C09120=1115.319,207.001,-67.010,-178.939,9.439,149.564
C09121=1115.314,207.249,-67.035,-178.936,9.442,149.564
C09122=1115.310,207.498,-67.061,-178.933,9.445,149.564
C09123=1115.306,207.747,-67.087,-178.930,9.447,149.564
C09124=1115.301,207.995,-67.112,-178.927,9.450,149.564
C09125=1115.297,208.244,-67.138,-178.925,9.453,149.564
C09126=1115.292,208.493,-67.164,-178.922,9.456,149.564
C09127=1115.288,208.741,-67.190,-178.919,9.459,149.564
C09128=1115.283,208.990,-67.215,-178.916,9.462,149.564
C09129=1115.279,209.238,-67.241,-178.914,9.465,149.564
C09130=1115.275,209.487,-67.266,-178.911,9.468,149.564
C09131=1115.271,209.736,-67.292,-178.908,9.470,149.564
C09132=1115.266,209.984,-67.318,-178.906,9.474,149.564
C09133=1115.262,210.233,-67.343,-178.903,9.476,149.564
C09134=1115.257,210.482,-67.370,-178.900,9.479,149.564
C09135=1115.252,210.731,-67.395,-178.897,9.482,149.563
C09136=1115.248,210.979,-67.421,-178.895,9.485,149.564
C09137=1115.244,211.227,-67.447,-178.892,9.488,149.564
C09138=1115.239,211.476,-67.473,-178.889,9.491,149.563
C09139=1115.235,211.725,-67.499,-178.887,9.494,149.564
C09140=1115.231,211.938,-67.521,-178.884,9.497,149.564
C09141=1115.227,212.151,-67.543,-178.882,9.499,149.563
C09142=1115.224,212.365,-67.565,-178.879,9.502,149.563
C09143=1115.220,212.579,-67.588,-178.877,9.505,149.564
C09144=1115.216,212.791,-67.609,-178.875,9.508,149.564
C09145=1115.212,213.005,-67.632,-178.873,9.510,149.564
C09146=1115.208,213.218,-67.654,-178.870,9.513,149.564
C09147=1115.204,213.432,-67.677,-178.869,9.516,149.564
C09148=1115.199,213.680,-67.703,-178.866,9.519,149.564
C09149=1115.196,213.928,-67.729,-178.864,9.521,149.564
C09150=1115.191,214.177,-67.755,-178.862,9.524,149.564
C09151=1115.187,214.426,-67.781,-178.860,9.527,149.564
C09152=1115.182,214.675,-67.807,-178.858,9.530,149.564
C09153=1115.178,214.923,-67.833,-178.856,9.532,149.564
C09154=1115.174,215.172,-67.859,-178.854,9.536,149.565
C09155=1115.168,215.420,-67.885,-178.851,9.539,149.565
C09156=1115.165,215.668,-67.912,-178.849,9.541,149.565
C09157=1115.160,215.917,-67.937,-178.847,9.544,149.565
C09158=1115.156,216.166,-67.963,-178.845,9.548,149.565
C09159=1115.151,216.415,-67.990,-178.843,9.550,149.565
C09160=1115.147,216.663,-68.016,-178.840,9.553,149.565
C09161=1115.143,216.912,-68.042,-178.838,9.556,149.565
C09162=1115.138,217.161,-68.069,-178.836,9.559,149.565
C09163=1115.134,217.409,-68.094,-178.834,9.562,149.565
C09164=1115.130,217.657,-68.121,-178.831,9.565,149.566
C09165=1115.125,217.906,-68.147,-178.829,9.568,149.566
C09166=1115.121,218.154,-68.173,-178.827,9.571,149.566
C09167=1115.116,218.403,-68.199,-178.825,9.574,149.566
C09168=1115.112,218.652,-68.226,-178.822,9.577,149.566
C09169=1115.108,218.900,-68.252,-178.819,9.580,149.566
C09170=1115.103,219.149,-68.279,-178.817,9.584,149.566
C09171=1115.099,219.398,-68.305,-178.815,9.587,149.566
C09172=1115.095,219.646,-68.331,-178.813,9.589,149.566
C09173=1115.090,219.895,-68.358,-178.810,9.593,149.566
C09174=1115.086,220.143,-68.384,-178.808,9.596,149.567
C09175=1115.081,220.392,-68.410,-178.805,9.599,149.567
C09176=1115.077,220.640,-68.437,-178.803,9.602,149.567
C09177=1115.072,220.889,-68.464,-178.801,9.605,149.567
C09178=1115.068,221.138,-68.490,-178.798,9.608,149.567
C09179=1115.063,221.386,-68.517,-178.796,9.612,149.567
C09180=1115.060,221.634,-68.543,-178.793,9.615,149.567
C09181=1115.055,221.884,-68.570,-178.791,9.618,149.567
C09182=1115.051,222.132,-68.596,-178.788,9.621,149.567
C09183=1115.046,222.380,-68.623,-178.786,9.624,149.567
C09184=1115.042,222.629,-68.649,-178.783,9.627,149.567
C09185=1115.037,222.877,-68.676,-178.781,9.630,149.567
C09186=1115.033,223.126,-68.702,-178.778,9.633,149.568
C09187=1115.028,223.375,-68.729,-178.775,9.636,149.568
C09188=1115.024,223.623,-68.755,-178.773,9.640,149.568
C09189=1115.020,223.871,-68.782,-178.770,9.643,149.568
C09190=1115.016,224.120,-68.809,-178.768,9.646,149.568
C09191=1115.011,224.369,-68.835,-178.765,9.649,149.568
C09192=1115.006,224.617,-68.862,-178.763,9.652,149.568
C09193=1115.002,224.865,-68.889,-178.760,9.655,149.568
C09194=1114.998,225.114,-68.916,-178.757,9.658,149.568
C09195=1114.994,225.362,-68.942,-178.755,9.661,149.568
C09196=1114.990,225.576,-68.965,-178.752,9.664,149.568
C09197=1114.986,225.789,-68.988,-178.750,9.666,149.568
C09198=1114.982,226.002,-69.011,-178.747,9.669,149.568
C09199=1114.979,226.215,-69.034,-178.746,9.671,149.568
C09200=1114.975,226.429,-69.057,-178.743,9.675,149.568
C09201=1114.971,226.642,-69.080,-178.741,9.678,149.568
C09202=1114.967,226.855,-69.103,-178.738,9.680,149.568
C09203=1114.963,227.068,-69.127,-178.736,9.683,149.568
C09204=1114.959,227.317,-69.153,-178.733,9.686,149.568
C09205=1114.955,227.565,-69.180,-178.730,9.689,149.568
C09206=1114.950,227.814,-69.207,-178.728,9.692,149.568
C09207=1114.946,228.062,-69.234,-178.725,9.694,149.568
C09208=1114.942,228.310,-69.261,-178.722,9.698,149.568
C09209=1114.937,228.560,-69.288,-178.719,9.701,149.568
C09210=1114.933,228.808,-69.315,-178.716,9.704,149.568
C09211=1114.929,229.056,-69.342,-178.713,9.707,149.568
C09212=1114.924,229.305,-69.369,-178.711,9.710,149.568
C09213=1114.920,229.553,-69.396,-178.707,9.714,149.568
C09214=1114.915,229.802,-69.423,-178.704,9.716,149.568
C09215=1114.912,230.051,-69.450,-178.701,9.719,149.568
C09216=1114.907,230.299,-69.477,-178.699,9.722,149.568
C09217=1114.902,230.548,-69.504,-178.695,9.726,149.568
C09218=1114.898,230.796,-69.531,-178.692,9.728,149.567
C09219=1114.893,231.044,-69.559,-178.689,9.731,149.567
C09220=1114.890,231.293,-69.586,-178.687,9.734,149.567
C09221=1114.885,231.541,-69.613,-178.684,9.737,149.567
C09222=1114.881,231.790,-69.640,-178.681,9.740,149.567
C09223=1114.876,232.038,-69.667,-178.678,9.743,149.567
C09224=1114.872,232.286,-69.695,-178.675,9.746,149.567
C09225=1114.868,232.535,-69.722,-178.672,9.748,149.567
C09226=1114.863,232.784,-69.749,-178.669,9.751,149.567
C09227=1114.858,233.032,-69.776,-178.666,9.754,149.567
C09228=1114.855,233.280,-69.803,-178.664,9.757,149.567
C09229=1114.851,233.529,-69.831,-178.661,9.759,149.566
C09230=1114.846,233.778,-69.858,-178.658,9.763,149.566
C09231=1114.841,234.026,-69.885,-178.655,9.765,149.566
C09232=1114.837,234.274,-69.913,-178.652,9.768,149.566
C09233=1114.833,234.523,-69.940,-178.649,9.771,149.566
C09234=1114.829,234.771,-69.968,-178.646,9.774,149.566
C09235=1114.824,235.020,-69.995,-178.643,9.776,149.566
C09236=1114.820,235.269,-70.022,-178.641,9.779,149.566
C09237=1114.815,235.517,-70.050,-178.638,9.781,149.566
C09238=1114.811,235.765,-70.077,-178.636,9.784,149.566
C09239=1114.807,236.014,-70.105,-178.633,9.787,149.566
C09240=1114.802,236.262,-70.132,-178.630,9.790,149.565
C09241=1114.798,236.511,-70.159,-178.627,9.792,149.565
C09242=1114.794,236.759,-70.188,-178.625,9.795,149.565
C09243=1114.789,237.008,-70.215,-178.622,9.797,149.565
C09244=1114.785,237.256,-70.242,-178.619,9.800,149.565
C09245=1114.781,237.505,-70.270,-178.617,9.802,149.565
C09246=1114.777,237.753,-70.298,-178.614,9.805,149.565
C09247=1114.772,238.001,-70.325,-178.611,9.808,149.565
C09248=1114.768,238.250,-70.353,-178.609,9.810,149.565
C09249=1114.764,238.498,-70.381,-178.606,9.813,149.565
C09250=1114.759,238.746,-70.408,-178.603,9.815,149.565
C09251=1114.755,238.995,-70.436,-178.601,9.818,149.565
C09252=1114.751,239.208,-70.460,-178.599,9.820,149.564
C09253=1114.747,239.421,-70.483,-178.596,9.822,149.564
C09254=1114.743,239.634,-70.507,-178.595,9.824,149.564
C09255=1114.740,239.847,-70.530,-178.592,9.827,149.564
C09256=1114.737,240.061,-70.554,-178.590,9.829,149.564
C09257=1114.732,240.274,-70.579,-178.587,9.831,149.564
C09258=1114.729,240.487,-70.603,-178.585,9.833,149.564
C09259=1114.725,240.700,-70.626,-178.583,9.835,149.564
C09260=1114.721,240.947,-70.654,-178.581,9.837,149.564
C09261=1114.717,241.197,-70.681,-178.578,9.841,149.564
C09262=1114.712,241.445,-70.709,-178.576,9.843,149.564
C09263=1114.708,241.693,-70.738,-178.573,9.846,149.564
C09264=1114.703,241.941,-70.766,-178.571,9.848,149.564
C09265=1114.699,242.191,-70.793,-178.569,9.851,149.564
C09266=1114.695,242.438,-70.821,-178.566,9.853,149.564
C09267=1114.691,242.686,-70.849,-178.564,9.856,149.564
C09268=1114.686,242.935,-70.877,-178.561,9.858,149.564
C09269=1114.681,243.184,-70.904,-178.559,9.861,149.564
C09270=1114.678,243.432,-70.932,-178.557,9.863,149.564
C09271=1114.673,243.680,-70.960,-178.554,9.866,149.564
C09272=1114.670,243.929,-70.988,-178.552,9.868,149.564
C09273=1114.665,244.177,-71.017,-178.550,9.870,149.564
C09274=1114.660,244.426,-71.044,-178.547,9.873,149.564
C09275=1114.656,244.674,-71.072,-178.545,9.876,149.564
C09276=1114.652,244.923,-71.101,-178.543,9.879,149.564
C09277=1114.647,245.171,-71.128,-178.541,9.881,149.564
C09278=1114.644,245.419,-71.157,-178.539,9.883,149.564
C09279=1114.639,245.667,-71.184,-178.536,9.886,149.564
C09280=1114.635,245.916,-71.213,-178.534,9.889,149.564
C09281=1114.630,246.164,-71.241,-178.532,9.891,149.564
C09282=1114.627,246.412,-71.269,-178.530,9.894,149.564
C09283=1114.621,246.661,-71.297,-178.528,9.896,149.564
C09284=1114.617,246.910,-71.325,-178.526,9.899,149.564
C09285=1114.613,247.158,-71.353,-178.524,9.902,149.564
C09286=1114.609,247.407,-71.381,-178.522,9.904,149.564
C09287=1114.604,247.655,-71.409,-178.518,9.908,149.564
C09288=1114.600,247.903,-71.438,-178.515,9.911,149.564
C09289=1114.595,248.151,-71.466,-178.510,9.915,149.564
C09290=1114.592,248.400,-71.494,-178.506,9.918,149.564
C09291=1114.588,248.648,-71.523,-178.502,9.923,149.563
C09292=1114.583,248.896,-71.551,-178.498,9.926,149.563
C09293=1114.579,249.145,-71.580,-178.494,9.929,149.563
C09294=1114.574,249.393,-71.608,-178.490,9.933,149.563
C09295=1114.571,249.641,-71.636,-178.486,9.936,149.563
C09296=1114.565,249.890,-71.664,-178.483,9.938,149.562
C09297=1114.562,250.138,-71.692,-178.479,9.942,149.562
C09298=1114.557,250.387,-71.721,-178.476,9.944,149.562
C09299=1114.553,250.634,-71.749,-178.472,9.948,149.562
C09300=1114.549,250.883,-71.778,-178.469,9.950,149.561
C09301=1114.545,251.132,-71.806,-178.466,9.953,149.561
C09302=1114.540,251.380,-71.835,-178.463,9.955,149.561
C09303=1114.536,251.628,-71.864,-178.460,9.958,149.561
C09304=1114.532,251.877,-71.892,-178.457,9.961,149.561
C09305=1114.528,252.125,-71.920,-178.453,9.963,149.560
C09306=1114.523,252.374,-71.949,-178.450,9.966,149.560
C09307=1114.519,252.622,-71.978,-178.448,9.968,149.560
C09308=1114.515,252.834,-72.002,-178.446,9.970,149.560
C09309=1114.511,253.048,-72.027,-178.444,9.972,149.560
C09310=1114.508,253.261,-72.051,-178.441,9.974,149.560
C09311=1114.504,253.473,-72.076,-178.439,9.976,149.560
C09312=1114.501,253.686,-72.100,-178.437,9.978,149.560
C09313=1114.497,253.899,-72.125,-178.435,9.979,149.560
C09314=1114.493,254.112,-72.149,-178.433,9.982,149.560
C09315=1114.490,254.326,-72.174,-178.432,9.983,149.560
C09316=1114.485,254.573,-72.203,-178.429,9.985,149.559
C09317=1114.481,254.822,-72.231,-178.428,9.987,149.559
C09318=1114.477,255.070,-72.261,-178.426,9.989,149.559
C09319=1114.472,255.318,-72.289,-178.424,9.992,149.560
C09320=1114.468,255.567,-72.317,-178.423,9.993,149.560
C09321=1114.464,255.815,-72.347,-178.421,9.996,149.560
C09322=1114.460,256.064,-72.375,-178.419,9.998,149.560
C09323=1114.455,256.311,-72.404,-178.416,10.000,149.560
C09324=1114.451,256.560,-72.433,-178.413,10.003,149.559
C09325=1114.447,256.808,-72.462,-178.411,10.006,149.560
C09326=1114.443,257.057,-72.490,-178.408,10.009,149.559
C09327=1114.438,257.304,-72.519,-178.405,10.011,149.559
C09328=1114.434,257.553,-72.548,-178.402,10.014,149.559
C09329=1114.430,257.801,-72.577,-178.399,10.017,149.559
C09330=1114.426,258.050,-72.606,-178.397,10.020,149.559
C09331=1114.421,258.298,-72.635,-178.394,10.023,149.559
C09332=1114.417,258.546,-72.664,-178.391,10.025,149.559
C09333=1114.413,258.795,-72.692,-178.388,10.028,149.559
C09334=1114.409,259.043,-72.722,-178.385,10.031,149.559
C09335=1114.404,259.291,-72.750,-178.382,10.034,149.559
C09336=1114.400,259.539,-72.780,-178.379,10.036,149.559
C09337=1114.396,259.787,-72.809,-178.377,10.040,149.559
C09338=1114.392,260.036,-72.837,-178.374,10.042,149.559
C09339=1114.388,260.284,-72.867,-178.371,10.045,149.558
C09340=1114.383,260.532,-72.896,-178.368,10.048,149.558
C09341=1114.378,260.781,-72.925,-178.365,10.051,149.558
C09342=1114.374,261.029,-72.954,-178.362,10.053,149.558
C09343=1114.371,261.277,-72.983,-178.359,10.056,149.558
C09344=1114.367,261.525,-73.012,-178.356,10.059,149.558
C09345=1114.362,261.774,-73.041,-178.353,10.061,149.558
C09346=1114.358,262.023,-73.070,-178.350,10.064,149.558
C09347=1114.353,262.270,-73.100,-178.347,10.067,149.557
C09348=1114.349,262.518,-73.129,-178.343,10.070,149.557
C09349=1114.345,262.767,-73.158,-178.340,10.073,149.557
C09350=1114.340,263.016,-73.187,-178.337,10.076,149.557
C09351=1114.337,263.263,-73.216,-178.334,10.078,149.557
C09352=1114.333,263.512,-73.246,-178.331,10.081,149.557
C09353=1114.328,263.760,-73.275,-178.328,10.084,149.557
C09354=1114.324,264.008,-73.304,-178.325,10.086,149.556
C09355=1114.319,264.256,-73.334,-178.322,10.089,149.556
C09356=1114.315,264.504,-73.363,-178.318,10.092,149.556
C09357=1114.311,264.752,-73.392,-178.316,10.094,149.556
C09358=1114.307,265.001,-73.422,-178.313,10.097,149.556
C09359=1114.303,265.249,-73.451,-178.310,10.100,149.556
C09360=1114.299,265.497,-73.481,-178.308,10.102,149.556
C09361=1114.294,265.745,-73.510,-178.304,10.104,149.555
C09362=1114.290,265.994,-73.540,-178.302,10.106,149.555
C09363=1114.286,266.242,-73.569,-178.299,10.109,149.555
C09364=1114.282,266.455,-73.594,-178.297,10.111,149.555
C09365=1114.278,266.668,-73.619,-178.295,10.113,149.555
C09366=1114.274,266.880,-73.645,-178.292,10.116,149.555
C09367=1114.271,267.094,-73.670,-178.290,10.118,149.555
C09368=1114.268,267.306,-73.696,-178.287,10.120,149.555
C09369=1114.263,267.519,-73.721,-178.285,10.122,149.555
C09370=1114.260,267.732,-73.746,-178.283,10.124,149.554
C09371=1114.256,267.945,-73.771,-178.280,10.127,149.554
C09372=1114.252,268.193,-73.801,-178.277,10.129,149.554
C09373=1114.248,268.441,-73.830,-178.275,10.132,149.554
C09374=1114.244,268.689,-73.860,-178.272,10.134,149.554
C09375=1114.240,268.937,-73.890,-178.269,10.137,149.554
C09376=1114.235,269.185,-73.919,-178.266,10.139,149.554
C09377=1114.231,269.434,-73.949,-178.263,10.142,149.554
C09378=1114.226,269.682,-73.979,-178.260,10.145,149.554
C09379=1114.222,269.930,-74.009,-178.258,10.147,149.554
C09380=1114.218,270.178,-74.038,-178.255,10.149,149.553
C09381=1114.214,270.426,-74.068,-178.252,10.152,149.553
C09382=1114.210,270.675,-74.098,-178.249,10.155,149.553
C09383=1114.206,270.924,-74.127,-178.246,10.158,149.553
C09384=1114.202,271.172,-74.158,-178.243,10.160,149.553
C09385=1114.197,271.420,-74.187,-178.241,10.162,149.553
C09386=1114.193,271.668,-74.217,-178.238,10.165,149.553
C09387=1114.189,271.916,-74.247,-178.235,10.168,149.553
C09388=1114.185,272.164,-74.276,-178.232,10.171,149.553
C09389=1114.180,272.413,-74.306,-178.229,10.173,149.553
C09390=1114.176,272.660,-74.337,-178.226,10.176,149.552
C09391=1114.172,272.908,-74.366,-178.224,10.179,149.552
C09392=1114.168,273.157,-74.396,-178.221,10.181,149.552
C09393=1114.163,273.405,-74.426,-178.218,10.184,149.552
C09394=1114.159,273.653,-74.456,-178.215,10.186,149.552
C09395=1114.155,273.901,-74.486,-178.212,10.189,149.552
C09396=1114.152,274.150,-74.516,-178.209,10.192,149.552
C09397=1114.147,274.398,-74.547,-178.206,10.194,149.552
C09398=1114.143,274.646,-74.576,-178.203,10.197,149.551
C09399=1114.139,274.893,-74.606,-178.200,10.200,149.551
C09400=1114.134,275.142,-74.636,-178.197,10.203,149.551
C09401=1114.130,275.390,-74.666,-178.194,10.205,149.551
C09402=1114.126,275.638,-74.696,-178.192,10.207,149.551
C09403=1114.122,275.887,-74.727,-178.189,10.210,149.551
C09404=1114.118,276.135,-74.756,-178.186,10.213,149.551
C09405=1114.114,276.383,-74.787,-178.183,10.215,149.551
C09406=1114.109,276.631,-74.817,-178.180,10.218,149.550
C09407=1114.105,276.879,-74.847,-178.177,10.221,149.550
C09408=1114.101,277.126,-74.877,-178.174,10.223,149.550
C09409=1114.097,277.376,-74.907,-178.171,10.226,149.550
C09410=1114.093,277.623,-74.938,-178.168,10.229,149.550
C09411=1114.088,277.872,-74.968,-178.164,10.231,149.550
C09412=1114.084,278.120,-74.998,-178.161,10.234,149.549
C09413=1114.081,278.367,-75.028,-178.159,10.237,149.549
C09414=1114.076,278.617,-75.058,-178.155,10.239,149.549
C09415=1114.072,278.864,-75.088,-178.152,10.242,149.549
C09416=1114.068,279.112,-75.119,-178.149,10.245,149.549
C09417=1114.064,279.360,-75.149,-178.146,10.247,149.549
C09418=1114.060,279.609,-75.180,-178.143,10.250,149.549
C09419=1114.056,279.857,-75.210,-178.140,10.253,149.548
C09420=1114.052,280.070,-75.237,-178.137,10.254,149.548
C09421=1114.048,280.282,-75.262,-178.134,10.257,149.548
C09422=1114.045,280.495,-75.288,-178.132,10.259,149.548
C09423=1114.041,280.708,-75.314,-178.129,10.262,149.548
C09424=1114.038,280.920,-75.341,-178.127,10.264,149.548
C09425=1114.034,281.133,-75.367,-178.124,10.266,149.547
C09426=1114.030,281.345,-75.393,-178.121,10.268,149.547
C09427=1114.027,281.558,-75.419,-178.119,10.270,149.547
C09428=1114.023,281.806,-75.449,-178.116,10.273,149.547
C09429=1114.019,282.054,-75.480,-178.113,10.275,149.547
C09430=1114.014,282.302,-75.511,-178.109,10.278,149.547
C09431=1114.010,282.550,-75.541,-178.106,10.281,149.546
C09432=1114.006,282.799,-75.572,-178.103,10.283,149.546
C09433=1114.002,283.047,-75.602,-178.100,10.286,149.546
C09434=1113.997,283.295,-75.633,-178.097,10.288,149.546
C09435=1113.993,283.543,-75.664,-178.094,10.290,149.546
C09436=1113.989,283.791,-75.694,-178.092,10.293,149.546
C09437=1113.985,284.039,-75.725,-178.089,10.296,149.545
C09438=1113.980,284.287,-75.755,-178.085,10.298,149.545
C09439=1113.977,284.535,-75.786,-178.082,10.301,149.545
C09440=1113.972,284.783,-75.817,-178.079,10.303,149.545
C09441=1113.968,285.031,-75.847,-178.076,10.306,149.545
C09442=1113.964,285.280,-75.878,-178.073,10.308,149.544
C09443=1113.960,285.527,-75.909,-178.070,10.311,149.544
C09444=1113.956,285.776,-75.941,-178.067,10.313,149.544
C09445=1113.952,286.023,-75.971,-178.064,10.316,149.544
C09446=1113.948,286.271,-76.001,-178.061,10.318,149.544
C09447=1113.944,286.520,-76.033,-178.058,10.321,149.544
C09448=1113.939,286.768,-76.063,-178.055,10.324,149.544
C09449=1113.935,287.015,-76.094,-178.052,10.326,149.543
C09450=1113.931,287.264,-76.125,-178.049,10.329,149.543
C09451=1113.927,287.511,-76.156,-178.046,10.331,149.543
C09452=1113.923,287.760,-76.187,-178.042,10.334,149.543
C09453=1113.919,288.008,-76.217,-178.040,10.336,149.543
C09454=1113.914,288.256,-76.248,-178.037,10.338,149.542
C09455=1113.911,288.504,-76.280,-178.034,10.341,149.542
C09456=1113.906,288.752,-76.311,-178.030,10.343,149.542
C09457=1113.902,289.000,-76.342,-178.028,10.346,149.542
C09458=1113.898,289.248,-76.372,-178.025,10.349,149.542
C09459=1113.894,289.496,-76.404,-178.021,10.351,149.542
C09460=1113.890,289.744,-76.435,-178.018,10.354,149.542
C09461=1113.886,289.993,-76.466,-178.015,10.357,149.541
C09462=1113.882,290.240,-76.497,-178.013,10.359,149.541
C09463=1113.877,290.489,-76.528,-178.009,10.361,149.541
C09464=1113.873,290.737,-76.559,-178.006,10.364,149.541
C09465=1113.869,290.984,-76.590,-178.003,10.366,149.540
C09466=1113.865,291.232,-76.621,-178.000,10.369,149.540
C09467=1113.861,291.480,-76.653,-177.997,10.371,149.540
C09468=1113.857,291.728,-76.684,-177.994,10.374,149.540
C09469=1113.852,291.976,-76.715,-177.991,10.377,149.540
C09470=1113.849,292.224,-76.746,-177.988,10.379,149.540
C09471=1113.844,292.472,-76.777,-177.985,10.381,149.540
C09472=1113.840,292.720,-76.809,-177.982,10.384,149.539
C09473=1113.836,292.969,-76.840,-177.979,10.387,149.539
C09474=1113.832,293.216,-76.872,-177.976,10.389,149.539
C09475=1113.828,293.465,-76.903,-177.973,10.392,149.539
C09476=1113.825,293.677,-76.929,-177.970,10.394,149.539
C09477=1113.821,293.890,-76.957,-177.967,10.396,149.538
C09478=1113.818,294.102,-76.984,-177.965,10.398,149.538
C09479=1113.814,294.315,-77.010,-177.963,10.400,149.538
C09480=1113.811,294.527,-77.037,-177.960,10.403,149.538
C09481=1113.807,294.740,-77.064,-177.957,10.405,149.538
C09482=1113.803,294.952,-77.091,-177.955,10.407,149.538
C09483=1113.800,295.164,-77.118,-177.952,10.409,149.538
C09484=1113.796,295.413,-77.149,-177.948,10.412,149.537
C09485=1113.792,295.660,-77.181,-177.946,10.414,149.537
C09486=1113.788,295.908,-77.212,-177.943,10.416,149.537
C09487=1113.783,296.157,-77.244,-177.940,10.419,149.537
C09488=1113.779,296.405,-77.276,-177.936,10.421,149.537
C09489=1113.776,296.653,-77.307,-177.933,10.424,149.537
C09490=1113.771,296.901,-77.338,-177.930,10.427,149.536
C09491=1113.767,297.149,-77.370,-177.927,10.429,149.536
C09492=1113.763,297.396,-77.402,-177.924,10.432,149.536
C09493=1113.759,297.644,-77.433,-177.921,10.435,149.536
C09494=1113.755,297.893,-77.465,-177.918,10.436,149.536
C09495=1113.751,298.140,-77.496,-177.915,10.439,149.536
C09496=1113.747,298.389,-77.528,-177.912,10.442,149.535
C09497=1113.742,298.636,-77.560,-177.909,10.444,149.535
C09498=1113.739,298.884,-77.592,-177.906,10.447,149.535
C09499=1113.734,299.133,-77.623,-177.903,10.449,149.535
C09500=1113.730,299.380,-77.654,-177.900,10.452,149.535
C09501=1113.726,299.628,-77.686,-177.897,10.455,149.534
C09502=1113.722,299.876,-77.719,-177.894,10.457,149.534
C09503=1113.718,300.124,-77.750,-177.890,10.460,149.534
C09504=1113.714,300.372,-77.782,-177.888,10.462,149.534
C09505=1113.710,300.620,-77.814,-177.885,10.464,149.534
C09506=1113.705,300.867,-77.846,-177.882,10.467,149.534
C09507=1113.702,301.115,-77.878,-177.878,10.469,149.533
C09508=1113.698,301.363,-77.910,-177.875,10.472,149.533
C09509=1113.694,301.611,-77.941,-177.872,10.475,149.533
C09510=1113.689,301.859,-77.974,-177.869,10.477,149.533
C09511=1113.685,302.107,-78.005,-177.866,10.480,149.533
C09512=1113.682,302.355,-78.037,-177.863,10.483,149.533
C09513=1113.677,302.603,-78.069,-177.860,10.485,149.532
C09514=1113.673,302.851,-78.101,-177.857,10.487,149.532
C09515=1113.669,303.099,-78.133,-177.854,10.489,149.532
C09516=1113.664,303.347,-78.165,-177.851,10.492,149.532
C09517=1113.660,303.595,-78.197,-177.848,10.495,149.532
C09518=1113.657,303.843,-78.229,-177.844,10.497,149.531
C09519=1113.652,304.091,-78.261,-177.841,10.500,149.531
C09520=1113.648,304.338,-78.293,-177.838,10.502,149.531
C09521=1113.644,304.586,-78.325,-177.835,10.505,149.531
C09522=1113.640,304.834,-78.358,-177.832,10.507,149.531
C09523=1113.636,305.082,-78.390,-177.830,10.509,149.531
C09524=1113.632,305.331,-78.422,-177.826,10.512,149.530
C09525=1113.628,305.578,-78.453,-177.823,10.515,149.530
C09526=1113.624,305.826,-78.485,-177.820,10.517,149.530
C09527=1113.620,306.074,-78.518,-177.817,10.520,149.530
C09528=1113.616,306.322,-78.550,-177.814,10.522,149.530
C09529=1113.612,306.570,-78.583,-177.811,10.525,149.530
C09530=1113.607,306.817,-78.614,-177.807,10.527,149.529
C09531=1113.603,307.065,-78.647,-177.804,10.530,149.529
C09532=1113.600,307.278,-78.675,-177.802,10.532,149.529
C09533=1113.597,307.490,-78.703,-177.799,10.534,149.529
C09534=1113.593,307.703,-78.730,-177.797,10.537,149.529
C09535=1113.589,307.915,-78.757,-177.794,10.538,149.529
C09536=1113.586,308.127,-78.785,-177.792,10.540,149.528
C09537=1113.583,308.340,-78.813,-177.789,10.543,149.528
C09538=1113.580,308.552,-78.841,-177.786,10.545,149.528
C09539=1113.575,308.765,-78.869,-177.784,10.547,149.528
C09540=1113.572,309.012,-78.901,-177.780,10.549,149.528
C09541=1113.567,309.261,-78.934,-177.777,10.552,149.528
C09542=1113.564,309.508,-78.966,-177.774,10.554,149.527
C09543=1113.559,309.756,-78.999,-177.771,10.557,149.527
C09544=1113.556,310.004,-79.030,-177.768,10.560,149.527
C09545=1113.551,310.251,-79.063,-177.765,10.562,149.527
C09546=1113.547,310.499,-79.095,-177.762,10.565,149.527
C09547=1113.543,310.747,-79.128,-177.759,10.568,149.527
C09548=1113.539,310.996,-79.161,-177.755,10.570,149.526
C09549=1113.535,311.243,-79.193,-177.753,10.572,149.526
C09550=1113.531,311.491,-79.226,-177.750,10.574,149.526
C09551=1113.527,311.739,-79.258,-177.746,10.577,149.526
C09552=1113.523,311.986,-79.291,-177.743,10.580,149.526
C09553=1113.519,312.235,-79.324,-177.740,10.582,149.525
C09554=1113.516,312.482,-79.356,-177.737,10.585,149.525
C09555=1113.511,312.731,-79.389,-177.734,10.587,149.525
C09556=1113.507,312.978,-79.422,-177.730,10.590,149.525
C09557=1113.504,313.226,-79.454,-177.728,10.593,149.525
C09558=1113.499,313.474,-79.487,-177.724,10.595,149.525
C09559=1113.495,313.722,-79.520,-177.722,10.597,149.524
C09560=1113.491,313.968,-79.552,-177.719,10.599,149.524
C09561=1113.487,314.217,-79.585,-177.716,10.602,149.524
C09562=1113.482,314.465,-79.618,-177.712,10.605,149.524
C09563=1113.478,314.712,-79.651,-177.709,10.607,149.524
C09564=1113.475,314.960,-79.684,-177.706,10.610,149.524
C09565=1113.470,315.208,-79.716,-177.703,10.612,149.523
C09566=1113.466,315.456,-79.749,-177.700,10.615,149.523
C09567=1113.463,315.703,-79.782,-177.697,10.617,149.523
C09568=1113.459,315.951,-79.815,-177.693,10.620,149.523
C09569=1113.455,316.200,-79.848,-177.690,10.623,149.523
C09570=1113.451,316.448,-79.881,-177.688,10.624,149.522
C09571=1113.447,316.695,-79.914,-177.685,10.627,149.522
C09572=1113.443,316.943,-79.947,-177.681,10.630,149.522
C09573=1113.439,317.191,-79.980,-177.678,10.632,149.522
C09574=1113.435,317.438,-80.013,-177.675,10.635,149.522
C09575=1113.431,317.686,-80.046,-177.672,10.637,149.521
C09576=1113.427,317.934,-80.079,-177.669,10.640,149.521
C09577=1113.423,318.182,-80.111,-177.665,10.642,149.521
C09578=1113.419,318.430,-80.144,-177.662,10.645,149.521
C09579=1113.415,318.677,-80.177,-177.659,10.648,149.521
C09580=1113.411,318.925,-80.210,-177.657,10.649,149.521
C09581=1113.406,319.173,-80.244,-177.654,10.652,149.520
C09582=1113.402,319.420,-80.277,-177.650,10.655,149.520
C09583=1113.399,319.669,-80.310,-177.647,10.657,149.520
C09584=1113.395,319.916,-80.343,-177.644,10.660,149.520
C09585=1113.391,320.164,-80.376,-177.641,10.662,149.520
C09586=1113.387,320.412,-80.409,-177.638,10.665,149.520
C09587=1113.383,320.660,-80.442,-177.634,10.667,149.519
C09588=1113.379,320.871,-80.472,-177.632,10.669,149.519
C09589=1113.376,321.084,-80.500,-177.629,10.671,149.519
C09590=1113.372,321.296,-80.528,-177.627,10.674,149.519
C09591=1113.369,321.508,-80.557,-177.624,10.676,149.519
C09592=1113.365,321.721,-80.585,-177.621,10.678,149.519
C09593=1113.362,321.933,-80.613,-177.619,10.680,149.518
C09594=1113.358,322.145,-80.642,-177.616,10.682,149.518
C09595=1113.356,322.357,-80.671,-177.613,10.685,149.518
C09596=1113.352,322.605,-80.704,-177.610,10.686,149.518
C09597=1113.348,322.853,-80.737,-177.607,10.689,149.518
C09598=1113.343,323.100,-80.770,-177.604,10.692,149.518
C09599=1113.340,323.349,-80.804,-177.601,10.694,149.517
C09600=1113.336,323.596,-80.838,-177.598,10.697,149.517
C09601=1113.332,323.844,-80.871,-177.595,10.699,149.517
C09602=1113.328,324.091,-80.904,-177.591,10.702,149.517
C09603=1113.324,324.339,-80.937,-177.588,10.705,149.517
C09604=1113.320,324.587,-80.972,-177.585,10.707,149.516
C09605=1113.316,324.835,-81.005,-177.582,10.709,149.516
C09606=1113.312,325.082,-81.038,-177.579,10.712,149.516
C09607=1113.308,325.330,-81.072,-177.576,10.714,149.516
C09608=1113.303,325.578,-81.106,-177.573,10.716,149.516
C09609=1113.300,325.826,-81.139,-177.570,10.719,149.516
C09610=1113.296,326.073,-81.173,-177.566,10.722,149.515
C09611=1113.292,326.321,-81.206,-177.563,10.724,149.515
C09612=1113.288,326.568,-81.240,-177.560,10.727,149.515
C09613=1113.285,326.816,-81.273,-177.557,10.729,149.515
C09614=1113.280,327.064,-81.307,-177.554,10.732,149.514
C09615=1113.276,327.311,-81.341,-177.551,10.734,149.514
C09616=1113.272,327.559,-81.374,-177.547,10.737,149.514
C09617=1113.269,327.807,-81.408,-177.544,10.739,149.514
C09618=1113.264,328.055,-81.442,-177.542,10.741,149.514
C09619=1113.261,328.302,-81.475,-177.538,10.744,149.514
C09620=1113.256,328.551,-81.510,-177.535,10.746,149.513
C09621=1113.252,328.798,-81.543,-177.532,10.749,149.513
C09622=1113.248,329.045,-81.577,-177.529,10.752,149.513
C09623=1113.244,329.293,-81.611,-177.526,10.754,149.513
C09624=1113.240,329.541,-81.645,-177.523,10.757,149.513
C09625=1113.236,329.788,-81.679,-177.519,10.759,149.513
C09626=1113.233,330.036,-81.712,-177.516,10.762,149.512
C09627=1113.229,330.284,-81.746,-177.513,10.764,149.512
C09628=1113.224,330.531,-81.780,-177.510,10.766,149.512
C09629=1113.220,330.779,-81.814,-177.507,10.769,149.512
C09630=1113.217,331.027,-81.848,-177.504,10.771,149.511
C09631=1113.212,331.274,-81.882,-177.501,10.774,149.511
C09632=1113.208,331.522,-81.915,-177.497,10.776,149.511
C09633=1113.205,331.770,-81.950,-177.494,10.779,149.511
C09634=1113.201,332.017,-81.984,-177.491,10.781,149.511
C09635=1113.197,332.264,-82.018,-177.488,10.784,149.511
C09636=1113.193,332.513,-82.051,-177.485,10.786,149.510
C09637=1113.189,332.760,-82.086,-177.481,10.789,149.510
C09638=1113.185,333.008,-82.120,-177.478,10.792,149.510
C09639=1113.182,333.255,-82.154,-177.476,10.793,149.510
C09640=1113.177,333.503,-82.188,-177.472,10.796,149.510
C09641=1113.173,333.751,-82.222,-177.469,10.798,149.510
C09642=1113.170,333.998,-82.256,-177.466,10.801,149.509
C09643=1113.166,334.246,-82.291,-177.463,10.803,149.509
C09644=1113.162,334.458,-82.320,-177.460,10.805,149.509
C09645=1113.159,334.670,-82.350,-177.457,10.808,149.509
C09646=1113.155,334.883,-82.378,-177.455,10.810,149.509
C09647=1113.152,335.094,-82.407,-177.452,10.812,149.508
C09648=1113.149,335.306,-82.437,-177.449,10.814,149.508
C09649=1113.146,335.519,-82.466,-177.447,10.816,149.508
C09650=1113.142,335.731,-82.496,-177.444,10.819,149.508
C09651=1113.139,335.942,-82.525,-177.441,10.820,149.508
C09652=1113.135,336.191,-82.560,-177.438,10.823,149.508
C09653=1113.130,336.438,-82.593,-177.435,10.826,149.507
C09654=1113.127,336.686,-82.627,-177.431,10.828,149.507
C09655=1113.123,336.934,-82.662,-177.428,10.831,149.507
C09656=1113.119,337.181,-82.696,-177.426,10.833,149.507
C09657=1113.115,337.428,-82.731,-177.423,10.835,149.507
C09658=1113.111,337.676,-82.766,-177.419,10.838,149.506
C09659=1113.107,337.923,-82.800,-177.416,10.840,149.506
C09660=1113.103,338.171,-82.835,-177.413,10.843,149.506
C09661=1113.100,338.419,-82.869,-177.410,10.845,149.506
C09662=1113.096,338.667,-82.903,-177.406,10.848,149.506
C09663=1113.092,338.914,-82.937,-177.403,10.850,149.505
C09664=1113.088,339.162,-82.972,-177.400,10.853,149.505
C09665=1113.083,339.409,-83.007,-177.397,10.855,149.505
C09666=1113.080,339.657,-83.041,-177.393,10.858,149.505
C09667=1113.075,339.905,-83.075,-177.391,10.859,149.505
C09668=1113.072,340.152,-83.111,-177.387,10.862,149.504
C09669=1113.068,340.399,-83.145,-177.385,10.865,149.504
C09670=1113.064,340.647,-83.180,-177.381,10.867,149.504
C09671=1113.059,340.895,-83.214,-177.378,10.870,149.504
C09672=1113.056,341.143,-83.248,-177.375,10.872,149.504
C09673=1113.052,341.389,-83.283,-177.372,10.875,149.504
C09674=1113.048,341.637,-83.318,-177.368,10.877,149.503
C09675=1113.044,341.885,-83.352,-177.365,10.880,149.503
C09676=1113.040,342.132,-83.388,-177.362,10.882,149.503
C09677=1113.036,342.380,-83.423,-177.359,10.884,149.503
C09678=1113.033,342.627,-83.456,-177.356,10.887,149.503
C09679=1113.029,342.875,-83.491,-177.353,10.889,149.502
C09680=1113.024,343.122,-83.526,-177.350,10.892,149.502
C09681=1113.020,343.370,-83.561,-177.346,10.894,149.502
C09682=1113.017,343.617,-83.596,-177.343,10.897,149.502
C09683=1113.013,343.865,-83.631,-177.340,10.899,149.502
C09684=1113.009,344.113,-83.666,-177.337,10.902,149.501
C09685=1113.005,344.360,-83.701,-177.333,10.904,149.501
C09686=1113.001,344.608,-83.736,-177.330,10.907,149.501
C09687=1112.998,344.855,-83.771,-177.327,10.909,149.501
C09688=1112.993,345.103,-83.805,-177.324,10.911,149.501
C09689=1112.990,345.350,-83.841,-177.321,10.914,149.500
C09690=1112.986,345.598,-83.875,-177.318,10.916,149.500
C09691=1112.981,345.845,-83.911,-177.314,10.919,149.500
C09692=1112.978,346.093,-83.945,-177.311,10.921,149.500
C09693=1112.974,346.340,-83.980,-177.308,10.923,149.499
C09694=1112.970,346.588,-84.015,-177.305,10.926,149.499
C09695=1112.966,346.835,-84.050,-177.302,10.929,149.499
C09696=1112.962,347.083,-84.085,-177.298,10.931,149.499
C09697=1112.958,347.330,-84.120,-177.295,10.934,149.499
C09698=1112.954,347.578,-84.156,-177.292,10.936,149.499
C09699=1112.950,347.826,-84.191,-177.289,10.938,149.498
C09700=1112.947,348.037,-84.221,-177.286,10.941,149.498
C09701=1112.944,348.249,-84.250,-177.283,10.942,149.498
C09702=1112.941,348.461,-84.281,-177.281,10.944,149.498
C09703=1112.937,348.673,-84.311,-177.278,10.947,149.498
C09704=1112.934,348.885,-84.341,-177.276,10.949,149.498
C09705=1112.931,349.097,-84.371,-177.272,10.951,149.497
C09706=1112.927,349.309,-84.402,-177.270,10.953,149.497
C09707=1112.924,349.521,-84.431,-177.267,10.955,149.497
C09708=1112.920,349.769,-84.467,-177.264,10.957,149.497
C09709=1112.916,350.016,-84.502,-177.261,10.960,149.497
C09710=1112.912,350.263,-84.537,-177.257,10.962,149.496
C09711=1112.908,350.511,-84.572,-177.254,10.965,149.496
C09712=1112.905,350.759,-84.608,-177.250,10.968,149.496
C09713=1112.901,351.006,-84.643,-177.247,10.970,149.496
C09714=1112.897,351.253,-84.679,-177.243,10.973,149.495
C09715=1112.893,351.500,-84.714,-177.240,10.975,149.495
C09716=1112.889,351.749,-84.749,-177.237,10.978,149.495
C09717=1112.885,351.996,-84.785,-177.234,10.980,149.495
C09718=1112.882,352.244,-84.820,-177.230,10.983,149.495
C09719=1112.877,352.490,-84.855,-177.227,10.985,149.494
C09720=1112.874,352.738,-84.891,-177.224,10.988,149.494
C09721=1112.870,352.985,-84.926,-177.220,10.990,149.494
C09722=1112.866,353.233,-84.962,-177.217,10.992,149.494
C09723=1112.863,353.480,-84.997,-177.213,10.995,149.493
C09724=1112.859,353.728,-85.033,-177.210,10.997,149.493
C09725=1112.854,353.975,-85.069,-177.207,11.000,149.493
C09726=1112.850,354.223,-85.104,-177.203,11.002,149.493
C09727=1112.847,354.470,-85.140,-177.200,11.005,149.492
C09728=1112.843,354.718,-85.175,-177.197,11.007,149.492
C09729=1112.839,354.965,-85.211,-177.193,11.010,149.492
C09730=1112.836,355.213,-85.247,-177.190,11.012,149.492
C09731=1112.832,355.460,-85.282,-177.186,11.014,149.491
C09732=1112.827,355.707,-85.318,-177.183,11.017,149.491
C09733=1112.823,355.955,-85.353,-177.180,11.019,149.491
C09734=1112.820,356.202,-85.389,-177.177,11.022,149.491
C09735=1112.816,356.449,-85.425,-177.173,11.024,149.490
C09736=1112.813,356.696,-85.461,-177.170,11.026,149.490
C09737=1112.808,356.944,-85.497,-177.166,11.029,149.490
C09738=1112.805,357.192,-85.532,-177.163,11.031,149.490
C09739=1112.801,357.439,-85.568,-177.160,11.034,149.489
C09740=1112.797,357.687,-85.604,-177.156,11.036,149.489
C09741=1112.794,357.934,-85.640,-177.153,11.038,149.489
C09742=1112.790,358.182,-85.676,-177.149,11.041,149.489
C09743=1112.786,358.429,-85.711,-177.146,11.043,149.488
C09744=1112.782,358.677,-85.747,-177.143,11.046,149.488
C09745=1112.778,358.923,-85.783,-177.139,11.048,149.488
C09746=1112.774,359.170,-85.819,-177.136,11.050,149.488
C09747=1112.770,359.418,-85.855,-177.132,11.053,149.487
C09748=1112.767,359.665,-85.891,-177.129,11.055,149.487
C09749=1112.763,359.913,-85.927,-177.126,11.058,149.487
C09750=1112.759,360.160,-85.963,-177.122,11.060,149.487
C09751=1112.756,360.407,-85.999,-177.119,11.063,149.486
C09752=1112.751,360.655,-86.035,-177.115,11.065,149.486
C09753=1112.748,360.902,-86.071,-177.112,11.067,149.486
C09754=1112.744,361.149,-86.107,-177.109,11.070,149.486
C09755=1112.740,361.396,-86.144,-177.105,11.072,149.485
C09756=1112.738,361.609,-86.174,-177.103,11.074,149.485
C09757=1112.734,361.821,-86.205,-177.100,11.076,149.485
C09758=1112.730,362.033,-86.236,-177.097,11.078,149.485
C09759=1112.728,362.244,-86.266,-177.094,11.080,149.484
C09760=1112.724,362.456,-86.298,-177.091,11.082,149.484
C09761=1112.721,362.668,-86.329,-177.088,11.084,149.484
C09762=1112.718,362.880,-86.360,-177.085,11.087,149.484
C09763=1112.715,363.092,-86.391,-177.083,11.088,149.484
C09764=1112.710,363.339,-86.427,-177.079,11.090,149.483
C09765=1112.707,363.586,-86.464,-177.076,11.093,149.483
C09766=1112.703,363.833,-86.499,-177.072,11.095,149.483
C09767=1112.699,364.081,-86.536,-177.069,11.098,149.483
C09768=1112.696,364.328,-86.572,-177.066,11.100,149.482
C09769=1112.692,364.575,-86.609,-177.062,11.102,149.482
C09770=1112.688,364.822,-86.645,-177.059,11.105,149.482
C09771=1112.684,365.071,-86.681,-177.055,11.107,149.482
C09772=1112.681,365.318,-86.718,-177.052,11.110,149.481
C09773=1112.677,365.565,-86.754,-177.049,11.112,149.481
C09774=1112.673,365.812,-86.790,-177.045,11.114,149.481
C09775=1112.669,366.059,-86.827,-177.042,11.117,149.481
C09776=1112.665,366.307,-86.864,-177.038,11.119,149.480
C09777=1112.662,366.553,-86.900,-177.035,11.122,149.480
C09778=1112.657,366.801,-86.936,-177.032,11.124,149.480
C09779=1112.654,367.048,-86.972,-177.028,11.127,149.480
C09780=1112.651,367.296,-87.010,-177.025,11.129,149.479
C09781=1112.646,367.543,-87.046,-177.022,11.131,149.479
C09782=1112.643,367.790,-87.083,-177.018,11.134,149.479
C09783=1112.639,368.038,-87.119,-177.015,11.136,149.479
C09784=1112.635,368.285,-87.155,-177.012,11.139,149.478
C09785=1112.631,368.532,-87.192,-177.008,11.141,149.478
C09786=1112.627,368.779,-87.229,-177.005,11.143,149.478
C09787=1112.624,369.027,-87.265,-177.002,11.145,149.478
C09788=1112.620,369.274,-87.302,-176.999,11.148,149.477
C09789=1112.616,369.521,-87.339,-176.995,11.150,149.477
C09790=1112.613,369.768,-87.375,-176.992,11.153,149.477
C09791=1112.609,370.015,-87.412,-176.989,11.155,149.477
C09792=1112.605,370.263,-87.450,-176.985,11.157,149.476
C09793=1112.602,370.510,-87.486,-176.982,11.160,149.476
C09794=1112.598,370.757,-87.523,-176.979,11.162,149.476
C09795=1112.594,371.004,-87.559,-176.975,11.165,149.476
C09796=1112.590,371.252,-87.597,-176.972,11.167,149.476
C09797=1112.587,371.499,-87.633,-176.969,11.170,149.475
C09798=1112.583,371.746,-87.670,-176.965,11.172,149.475
C09799=1112.579,371.994,-87.707,-176.962,11.175,149.475
C09800=1112.575,372.241,-87.744,-176.959,11.177,149.475
C09801=1112.572,372.488,-87.780,-176.955,11.180,149.475
C09802=1112.568,372.736,-87.817,-176.952,11.182,149.474
C09803=1112.564,372.983,-87.854,-176.948,11.184,149.474
C09804=1112.560,373.231,-87.891,-176.945,11.187,149.474
C09805=1112.557,373.477,-87.928,-176.942,11.189,149.474
C09806=1112.553,373.724,-87.965,-176.939,11.192,149.473
C09807=1112.549,373.971,-88.002,-176.935,11.194,149.473
C09808=1112.545,374.219,-88.039,-176.932,11.197,149.473
C09809=1112.541,374.466,-88.076,-176.929,11.199,149.473
C09810=1112.538,374.713,-88.113,-176.925,11.202,149.473
C09811=1112.535,374.960,-88.150,-176.922,11.204,149.472
C09812=1112.531,375.172,-88.182,-176.919,11.207,149.472
C09813=1112.527,375.383,-88.214,-176.917,11.209,149.472
C09814=1112.525,375.595,-88.246,-176.913,11.211,149.472
C09815=1112.521,375.807,-88.278,-176.911,11.213,149.472
C09816=1112.518,376.019,-88.309,-176.908,11.216,149.472
C09817=1112.515,376.231,-88.340,-176.905,11.217,149.471
C09818=1112.512,376.442,-88.372,-176.902,11.220,149.471
C09819=1112.509,376.654,-88.404,-176.899,11.222,149.471
C09820=1112.505,376.901,-88.442,-176.896,11.224,149.471
C09821=1112.502,377.149,-88.479,-176.893,11.227,149.471
C09822=1112.498,377.395,-88.516,-176.890,11.229,149.471
C09823=1112.494,377.642,-88.553,-176.886,11.232,149.470
C09824=1112.490,377.890,-88.591,-176.883,11.234,149.470
C09825=1112.486,378.137,-88.628,-176.880,11.237,149.470
C09826=1112.482,378.384,-88.665,-176.877,11.239,149.470
C09827=1112.479,378.631,-88.703,-176.873,11.243,149.470
C09828=1112.475,378.878,-88.740,-176.870,11.245,149.470
C09829=1112.472,379.126,-88.778,-176.866,11.248,149.469
C09830=1112.468,379.373,-88.815,-176.863,11.251,149.469
C09831=1112.464,379.619,-88.852,-176.860,11.253,149.469
C09832=1112.460,379.867,-88.889,-176.857,11.256,149.469
C09833=1112.457,380.114,-88.927,-176.853,11.258,149.469
C09834=1112.453,380.361,-88.965,-176.851,11.261,149.469
C09835=1112.449,380.608,-89.002,-176.847,11.263,149.469
C09836=1112.445,380.855,-89.040,-176.844,11.266,149.468
C09837=1112.441,381.103,-89.077,-176.841,11.268,149.468
C09838=1112.438,381.350,-89.115,-176.838,11.271,149.468
C09839=1112.434,381.597,-89.153,-176.834,11.274,149.468
C09840=1112.430,381.844,-89.189,-176.831,11.277,149.468
C09841=1112.427,382.091,-89.227,-176.828,11.280,149.468
C09842=1112.423,382.338,-89.265,-176.824,11.282,149.468
C09843=1112.420,382.586,-89.302,-176.821,11.285,149.467
C09844=1112.416,382.832,-89.340,-176.818,11.287,149.467
C09845=1112.412,383.080,-89.378,-176.815,11.290,149.467
C09846=1112.408,383.327,-89.416,-176.812,11.293,149.467
C09847=1112.405,383.575,-89.453,-176.809,11.295,149.467
C09848=1112.401,383.821,-89.491,-176.806,11.298,149.467
C09849=1112.398,384.068,-89.529,-176.804,11.300,149.467
C09850=1112.394,384.315,-89.566,-176.801,11.303,149.467
C09851=1112.390,384.562,-89.605,-176.798,11.306,149.467
C09852=1112.386,384.810,-89.642,-176.796,11.308,149.467
C09853=1112.383,385.057,-89.680,-176.793,11.311,149.467
C09854=1112.379,385.304,-89.717,-176.790,11.313,149.467
C09855=1112.375,385.551,-89.756,-176.787,11.315,149.467
C09856=1112.371,385.798,-89.793,-176.785,11.319,149.467
C09857=1112.368,386.045,-89.831,-176.782,11.321,149.467
C09858=1112.365,386.292,-89.869,-176.780,11.323,149.467
C09859=1112.361,386.539,-89.907,-176.777,11.326,149.467
C09860=1112.357,386.786,-89.945,-176.774,11.329,149.467
C09861=1112.353,387.033,-89.983,-176.772,11.331,149.467
C09862=1112.350,387.280,-90.021,-176.769,11.334,149.467
C09863=1112.346,387.527,-90.059,-176.767,11.337,149.467
C09864=1112.343,387.774,-90.097,-176.764,11.340,149.467
C09865=1112.339,388.022,-90.135,-176.761,11.343,149.467
C09866=1112.336,388.268,-90.172,-176.759,11.345,149.467
C09867=1112.332,388.516,-90.211,-176.757,11.349,149.468
C09868=1112.328,388.727,-90.243,-176.754,11.351,149.467
C09869=1112.325,388.939,-90.276,-176.752,11.354,149.468
C09870=1112.322,389.151,-90.308,-176.750,11.356,149.468
C09871=1112.319,389.362,-90.341,-176.748,11.358,149.468
C09872=1112.316,389.573,-90.373,-176.745,11.361,149.468
C09873=1112.313,389.786,-90.406,-176.743,11.364,149.468
C09874=1112.310,389.996,-90.438,-176.741,11.366,149.468
C09875=1112.307,390.208,-90.472,-176.739,11.369,149.468
C09876=1112.303,390.455,-90.509,-176.736,11.372,149.469
C09877=1112.300,390.702,-90.547,-176.734,11.375,149.469
C09878=1112.296,390.949,-90.586,-176.731,11.379,149.469
C09879=1112.292,391.196,-90.623,-176.729,11.382,149.469
C09880=1112.289,391.443,-90.662,-176.726,11.385,149.469
C09881=1112.285,391.690,-90.700,-176.724,11.388,149.469
C09882=1112.281,391.937,-90.738,-176.721,11.391,149.470
C09883=1112.277,392.184,-90.777,-176.719,11.394,149.470
C09884=1112.274,392.431,-90.815,-176.716,11.397,149.470
C09885=1112.270,392.678,-90.853,-176.714,11.401,149.470
C09886=1112.267,392.925,-90.891,-176.712,11.404,149.471
C09887=1112.263,393.173,-90.930,-176.709,11.407,149.471
C09888=1112.260,393.419,-90.969,-176.707,11.410,149.471
C09889=1112.256,393.666,-91.006,-176.704,11.415,149.471
C09890=1112.252,393.914,-91.045,-176.702,11.418,149.472
C09891=1112.249,394.161,-91.084,-176.699,11.421,149.472
C09892=1112.245,394.407,-91.121,-176.697,11.424,149.472
C09893=1112.241,394.655,-91.160,-176.695,11.428,149.472
C09894=1112.238,394.901,-91.199,-176.692,11.432,149.473
C09895=1112.234,395.149,-91.237,-176.690,11.435,149.473
C09896=1112.231,395.395,-91.276,-176.688,11.439,149.473
C09897=1112.227,395.642,-91.314,-176.685,11.442,149.474
C09898=1112.224,395.890,-91.352,-176.682,11.446,149.474
C09899=1112.220,396.137,-91.391,-176.680,11.450,149.474
C09900=1112.216,396.383,-91.429,-176.678,11.453,149.475
C09901=1112.212,396.630,-91.468,-176.675,11.457,149.475
C09902=1112.209,396.878,-91.507,-176.673,11.461,149.476
C09903=1112.206,397.124,-91.545,-176.671,11.464,149.476
C09904=1112.201,397.371,-91.583,-176.668,11.469,149.476
C09905=1112.198,397.618,-91.622,-176.666,11.472,149.477
C09906=1112.195,397.865,-91.661,-176.664,11.477,149.477
C09907=1112.191,398.112,-91.700,-176.662,11.480,149.478
C09908=1112.188,398.359,-91.739,-176.659,11.484,149.478
C09909=1112.183,398.606,-91.777,-176.657,11.488,149.479
C09910=1112.180,398.853,-91.816,-176.655,11.492,149.479
C09911=1112.177,399.100,-91.855,-176.653,11.496,149.480
C09912=1112.173,399.347,-91.893,-176.650,11.500,149.480
C09913=1112.169,399.594,-91.932,-176.648,11.504,149.480
C09914=1112.166,399.840,-91.971,-176.646,11.508,149.481
C09915=1112.162,400.088,-92.009,-176.644,11.512,149.482
C09916=1112.158,400.335,-92.048,-176.641,11.517,149.482
C09917=1112.155,400.581,-92.087,-176.639,11.521,149.483
C09918=1112.151,400.829,-92.126,-176.637,11.525,149.483
C09919=1112.148,401.076,-92.165,-176.635,11.530,149.484
C09920=1112.144,401.323,-92.204,-176.633,11.534,149.484
C09921=1112.141,401.569,-92.242,-176.631,11.538,149.485
C09922=1112.137,401.816,-92.281,-176.628,11.542,149.486
C09923=1112.133,402.063,-92.320,-176.626,11.547,149.486
C09924=1112.130,402.274,-92.354,-176.624,11.551,149.487
C09925=1112.128,402.486,-92.387,-176.622,11.554,149.487
C09926=1112.125,402.698,-92.420,-176.621,11.558,149.488
C09927=1112.121,402.909,-92.453,-176.619,11.562,149.488
C09928=1112.118,403.120,-92.487,-176.617,11.566,149.489
C09929=1112.115,403.331,-92.520,-176.615,11.569,149.489
C09930=1112.112,403.543,-92.554,-176.613,11.574,149.490
C09931=1112.110,403.754,-92.587,-176.611,11.578,149.491
C09932=1112.106,404.001,-92.626,-176.609,11.583,149.491
C09933=1112.102,404.248,-92.666,-176.607,11.587,149.492
C09934=1112.099,404.495,-92.705,-176.606,11.591,149.493
C09935=1112.095,404.742,-92.744,-176.604,11.596,149.493
C09936=1112.092,404.989,-92.783,-176.601,11.601,149.494
C09937=1112.088,405.236,-92.823,-176.599,11.606,149.495
C09938=1112.084,405.482,-92.861,-176.597,11.611,149.496
C09939=1112.081,405.728,-92.900,-176.595,11.616,149.496
C09940=1112.077,405.975,-92.939,-176.594,11.621,149.497
C09941=1112.074,406.222,-92.979,-176.591,11.626,149.498
C09942=1112.070,406.469,-93.018,-176.589,11.631,149.499
C09943=1112.066,406.716,-93.057,-176.587,11.636,149.500
C09944=1112.063,406.963,-93.096,-176.585,11.641,149.500
C09945=1112.059,407.210,-93.136,-176.583,11.646,149.501
C09946=1112.055,407.457,-93.175,-176.582,11.651,149.502
C09947=1112.052,407.704,-93.214,-176.580,11.656,149.503
C09948=1112.049,407.951,-93.254,-176.577,11.662,149.504
C09949=1112.046,408.198,-93.293,-176.575,11.667,149.505
C09950=1112.043,408.445,-93.332,-176.573,11.672,149.506
C09951=1112.039,408.692,-93.372,-176.572,11.677,149.507
C09952=1112.035,408.939,-93.411,-176.570,11.683,149.508
C09953=1112.032,409.185,-93.451,-176.568,11.688,149.508
C09954=1112.028,409.432,-93.490,-176.566,11.693,149.509
C09955=1112.025,409.679,-93.529,-176.564,11.699,149.510
C09956=1112.022,409.925,-93.569,-176.562,11.704,149.511
C09957=1112.017,410.173,-93.609,-176.561,11.710,149.512
C09958=1112.014,410.420,-93.649,-176.559,11.716,149.513
C09959=1112.010,410.666,-93.688,-176.557,11.721,149.514
C09960=1112.007,410.913,-93.728,-176.555,11.727,149.515
C09961=1112.003,411.160,-93.767,-176.554,11.732,149.516
C09962=1112.000,411.406,-93.807,-176.551,11.738,149.518
C09963=1111.996,411.653,-93.846,-176.550,11.744,149.518
C09964=1111.993,411.901,-93.886,-176.548,11.750,149.520
C09965=1111.990,412.147,-93.926,-176.546,11.755,149.521
C09966=1111.986,412.394,-93.965,-176.544,11.762,149.522
C09967=1111.983,412.640,-94.005,-176.542,11.768,149.523
C09968=1111.978,412.888,-94.045,-176.541,11.773,149.524
C09969=1111.975,413.134,-94.085,-176.539,11.779,149.525
C09970=1111.972,413.381,-94.124,-176.537,11.786,149.526
C09971=1111.969,413.628,-94.164,-176.536,11.791,149.528
C09972=1111.966,413.874,-94.204,-176.534,11.798,149.529
C09973=1111.964,414.121,-94.243,-176.533,11.804,149.530
C09974=1111.963,414.369,-94.283,-176.531,11.809,149.531
C09975=1111.961,414.615,-94.322,-176.529,11.816,149.532
C09976=1111.961,414.862,-94.362,-176.528,11.822,149.534
C09977=1111.960,415.109,-94.402,-176.526,11.829,149.535
C09978=1111.960,415.356,-94.441,-176.525,11.834,149.536
C09979=1111.962,415.602,-94.480,-176.524,11.841,149.538
C09980=1111.963,415.813,-94.514,-176.522,11.846,149.538
C09981=1111.965,416.025,-94.547,-176.521,11.852,149.540
C09982=1111.966,416.236,-94.581,-176.519,11.857,149.541
C09983=1111.969,416.447,-94.614,-176.518,11.863,149.542
C09984=1111.971,416.658,-94.647,-176.517,11.868,149.543
C09985=1111.975,416.870,-94.680,-176.516,11.874,149.544
C09986=1111.978,417.080,-94.714,-176.515,11.879,149.545
C09987=1111.982,417.292,-94.747,-176.513,11.885,149.547
C09988=1111.563,417.291,-94.811,-176.506,11.889,149.546
C09989=1111.559,417.080,-94.777,-176.507,11.884,149.545
C09990=1111.556,416.868,-94.744,-176.508,11.878,149.544
C09991=1111.552,416.658,-94.710,-176.510,11.873,149.542
C09992=1111.550,416.447,-94.676,-176.511,11.867,149.541
C09993=1111.548,416.235,-94.643,-176.512,11.862,149.540
C09994=1111.546,416.025,-94.610,-176.513,11.856,149.539
C09995=1111.544,415.813,-94.576,-176.515,11.851,149.538
C09996=1111.543,415.602,-94.543,-176.516,11.845,149.537
//INST
///DATE 2021/06/15 17:29
///ATTR SC,RW,RJ
////FRAME ROBOT
///GROUP1 RB1
NOP
MOVL C00000 V=800.0 PL=0
MOVL C00001 V=800.0 PL=0
MOVL C00002 V=800.0 PL=0
MOVL C00003 V=800.0 PL=0
MOVL C00004 V=800.0 PL=0
MOVL C00005 V=800.0 PL=0
MOVL C00006 V=800.0 PL=0
MOVL C00007 V=800.0 PL=0
MOVL C00008 V=800.0 PL=0
MOVL C00009 V=800.0 PL=0
MOVL C00010 V=800.0 PL=0
MOVL C00011 V=800.0 PL=0
MOVL C00012 V=800.0 PL=0
MOVL C00013 V=800.0 PL=0
MOVL C00014 V=800.0 PL=0
MOVL C00015 V=800.0 PL=0
MOVL C00016 V=800.0 PL=0
MOVL C00017 V=800.0 PL=0
MOVL C00018 V=800.0 PL=0
MOVL C00019 V=800.0 PL=0
MOVL C00020 V=800.0 PL=0
MOVL C00021 V=800.0 PL=0
MOVL C00022 V=800.0 PL=0
MOVL C00023 V=800.0 PL=0
MOVL C00024 V=800.0 PL=0
MOVL C00025 V=800.0 PL=0
MOVL C00026 V=800.0 PL=0
MOVL C00027 V=800.0 PL=0
MOVL C00028 V=800.0 PL=0
MOVL C00029 V=800.0 PL=0
MOVL C00030 V=800.0 PL=0
MOVL C00031 V=800.0 PL=0
MOVL C00032 V=800.0 PL=0
MOVL C00033 V=800.0 PL=0
MOVL C00034 V=800.0 PL=0
MOVL C00035 V=800.0 PL=0
MOVL C00036 V=800.0 PL=0
MOVL C00037 V=800.0 PL=0
MOVL C00038 V=800.0 PL=0
MOVL C00039 V=800.0 PL=0
MOVL C00040 V=800.0 PL=0
MOVL C00041 V=800.0 PL=0
MOVL C00042 V=800.0 PL=0
MOVL C00043 V=800.0 PL=0
MOVL C00044 V=800.0 PL=0
MOVL C00045 V=800.0 PL=0
MOVL C00046 V=800.0 PL=0
MOVL C00047 V=800.0 PL=0
MOVL C00048 V=800.0 PL=0
MOVL C00049 V=800.0 PL=0
MOVL C00050 V=800.0 PL=0
MOVL C00051 V=800.0 PL=0
MOVL C00052 V=800.0 PL=0
MOVL C00053 V=800.0 PL=0
MOVL C00054 V=800.0 PL=0
MOVL C00055 V=800.0 PL=0
MOVL C00056 V=800.0 PL=0
MOVL C00057 V=800.0 PL=0
MOVL C00058 V=800.0 PL=0
MOVL C00059 V=800.0 PL=0
MOVL C00060 V=800.0 PL=0
MOVL C00061 V=800.0 PL=0
MOVL C00062 V=800.0 PL=0
MOVL C00063 V=800.0 PL=0
MOVL C00064 V=800.0 PL=0
MOVL C00065 V=800.0 PL=0
MOVL C00066 V=800.0 PL=0
MOVL C00067 V=800.0 PL=0
MOVL C00068 V=800.0 PL=0
MOVL C00069 V=800.0 PL=0
MOVL C00070 V=800.0 PL=0
MOVL C00071 V=800.0 PL=0
MOVL C00072 V=800.0 PL=0
MOVL C00073 V=800.0 PL=0
MOVL C00074 V=800.0 PL=0
MOVL C00075 V=800.0 PL=0
MOVL C00076 V=800.0 PL=0
MOVL C00077 V=800.0 PL=0
MOVL C00078 V=800.0 PL=0
MOVL C00079 V=800.0 PL=0
MOVL C00080 V=800.0 PL=0
MOVL C00081 V=800.0 PL=0
MOVL C00082 V=800.0 PL=0
MOVL C00083 V=800.0 PL=0
MOVL C00084 V=800.0 PL=0
MOVL C00085 V=800.0 PL=0
MOVL C00086 V=800.0 PL=0
MOVL C00087 V=800.0 PL=0
MOVL C00088 V=800.0 PL=0
MOVL C00089 V=800.0 PL=0
MOVL C00090 V=800.0 PL=0
MOVL C00091 V=800.0 PL=0
MOVL C00092 V=800.0 PL=0
MOVL C00093 V=800.0 PL=0
MOVL C00094 V=800.0 PL=0
MOVL C00095 V=800.0 PL=0
MOVL C00096 V=800.0 PL=0
MOVL C00097 V=800.0 PL=0
MOVL C00098 V=800.0 PL=0
MOVL C00099 V=800.0 PL=0
MOVL C00100 V=800.0 PL=0
MOVL C00101 V=800.0 PL=0
MOVL C00102 V=800.0 PL=0
MOVL C00103 V=800.0 PL=0
MOVL C00104 V=800.0 PL=0
MOVL C00105 V=800.0 PL=0
MOVL C00106 V=800.0 PL=0
MOVL C00107 V=800.0 PL=0
MOVL C00108 V=800.0 PL=0
MOVL C00109 V=800.0 PL=0
MOVL C00110 V=800.0 PL=0
MOVL C00111 V=800.0 PL=0
MOVL C00112 V=800.0 PL=0
MOVL C00113 V=800.0 PL=0
MOVL C00114 V=800.0 PL=0
MOVL C00115 V=800.0 PL=0
MOVL C00116 V=800.0 PL=0
MOVL C00117 V=800.0 PL=0
MOVL C00118 V=800.0 PL=0
MOVL C00119 V=800.0 PL=0
MOVL C00120 V=800.0 PL=0
MOVL C00121 V=800.0 PL=0
MOVL C00122 V=800.0 PL=0
MOVL C00123 V=800.0 PL=0
MOVL C00124 V=800.0 PL=0
MOVL C00125 V=800.0 PL=0
MOVL C00126 V=800.0 PL=0
MOVL C00127 V=800.0 PL=0
MOVL C00128 V=800.0 PL=0
MOVL C00129 V=800.0 PL=0
MOVL C00130 V=800.0 PL=0
MOVL C00131 V=800.0 PL=0
MOVL C00132 V=800.0 PL=0
MOVL C00133 V=800.0 PL=0
MOVL C00134 V=800.0 PL=0
MOVL C00135 V=800.0 PL=0
MOVL C00136 V=800.0 PL=0
MOVL C00137 V=800.0 PL=0
MOVL C00138 V=800.0 PL=0
MOVL C00139 V=800.0 PL=0
MOVL C00140 V=800.0 PL=0
MOVL C00141 V=800.0 PL=0
MOVL C00142 V=800.0 PL=0
MOVL C00143 V=800.0 PL=0
MOVL C00144 V=800.0 PL=0
MOVL C00145 V=800.0 PL=0
MOVL C00146 V=800.0 PL=0
MOVL C00147 V=800.0 PL=0
MOVL C00148 V=800.0 PL=0
MOVL C00149 V=800.0 PL=0
MOVL C00150 V=800.0 PL=0
MOVL C00151 V=800.0 PL=0
MOVL C00152 V=800.0 PL=0
MOVL C00153 V=800.0 PL=0
MOVL C00154 V=800.0 PL=0
MOVL C00155 V=800.0 PL=0
MOVL C00156 V=800.0 PL=0
MOVL C00157 V=800.0 PL=0
MOVL C00158 V=800.0 PL=0
MOVL C00159 V=800.0 PL=0
MOVL C00160 V=800.0 PL=0
MOVL C00161 V=800.0 PL=0
MOVL C00162 V=800.0 PL=0
MOVL C00163 V=800.0 PL=0
MOVL C00164 V=800.0 PL=0
MOVL C00165 V=800.0 PL=0
MOVL C00166 V=800.0 PL=0
MOVL C00167 V=800.0 PL=0
MOVL C00168 V=800.0 PL=0
MOVL C00169 V=800.0 PL=0
MOVL C00170 V=800.0 PL=0
MOVL C00171 V=800.0 PL=0
MOVL C00172 V=800.0 PL=0
MOVL C00173 V=800.0 PL=0
MOVL C00174 V=800.0 PL=0
MOVL C00175 V=800.0 PL=0
MOVL C00176 V=800.0 PL=0
MOVL C00177 V=800.0 PL=0
MOVL C00178 V=800.0 PL=0
MOVL C00179 V=800.0 PL=0
MOVL C00180 V=800.0 PL=0
MOVL C00181 V=800.0 PL=0
MOVL C00182 V=800.0 PL=0
MOVL C00183 V=800.0 PL=0
MOVL C00184 V=800.0 PL=0
MOVL C00185 V=800.0 PL=0
MOVL C00186 V=800.0 PL=0
MOVL C00187 V=800.0 PL=0
MOVL C00188 V=800.0 PL=0
MOVL C00189 V=800.0 PL=0
MOVL C00190 V=800.0 PL=0
MOVL C00191 V=800.0 PL=0
MOVL C00192 V=800.0 PL=0
MOVL C00193 V=800.0 PL=0
MOVL C00194 V=800.0 PL=0
MOVL C00195 V=800.0 PL=0
MOVL C00196 V=800.0 PL=0
MOVL C00197 V=800.0 PL=0
MOVL C00198 V=800.0 PL=0
MOVL C00199 V=800.0 PL=0
MOVL C00200 V=800.0 PL=0
MOVL C00201 V=800.0 PL=0
MOVL C00202 V=800.0 PL=0
MOVL C00203 V=800.0 PL=0
MOVL C00204 V=800.0 PL=0
MOVL C00205 V=800.0 PL=0
MOVL C00206 V=800.0 PL=0
MOVL C00207 V=800.0 PL=0
MOVL C00208 V=800.0 PL=0
MOVL C00209 V=800.0 PL=0
MOVL C00210 V=800.0 PL=0
MOVL C00211 V=800.0 PL=0
MOVL C00212 V=800.0 PL=0
MOVL C00213 V=800.0 PL=0
MOVL C00214 V=800.0 PL=0
MOVL C00215 V=800.0 PL=0
MOVL C00216 V=800.0 PL=0
MOVL C00217 V=800.0 PL=0
MOVL C00218 V=800.0 PL=0
MOVL C00219 V=800.0 PL=0
MOVL C00220 V=800.0 PL=0
MOVL C00221 V=800.0 PL=0
MOVL C00222 V=800.0 PL=0
MOVL C00223 V=800.0 PL=0
MOVL C00224 V=800.0 PL=0
MOVL C00225 V=800.0 PL=0
MOVL C00226 V=800.0 PL=0
MOVL C00227 V=800.0 PL=0
MOVL C00228 V=800.0 PL=0
MOVL C00229 V=800.0 PL=0
MOVL C00230 V=800.0 PL=0
MOVL C00231 V=800.0 PL=0
MOVL C00232 V=800.0 PL=0
MOVL C00233 V=800.0 PL=0
MOVL C00234 V=800.0 PL=0
MOVL C00235 V=800.0 PL=0
MOVL C00236 V=800.0 PL=0
MOVL C00237 V=800.0 PL=0
MOVL C00238 V=800.0 PL=0
MOVL C00239 V=800.0 PL=0
MOVL C00240 V=800.0 PL=0
MOVL C00241 V=800.0 PL=0
MOVL C00242 V=800.0 PL=0
MOVL C00243 V=800.0 PL=0
MOVL C00244 V=800.0 PL=0
MOVL C00245 V=800.0 PL=0
MOVL C00246 V=800.0 PL=0
MOVL C00247 V=800.0 PL=0
MOVL C00248 V=800.0 PL=0
MOVL C00249 V=800.0 PL=0
MOVL C00250 V=800.0 PL=0
MOVL C00251 V=800.0 PL=0
MOVL C00252 V=800.0 PL=0
MOVL C00253 V=800.0 PL=0
MOVL C00254 V=800.0 PL=0
MOVL C00255 V=800.0 PL=0
MOVL C00256 V=800.0 PL=0
MOVL C00257 V=800.0 PL=0
MOVL C00258 V=800.0 PL=0
MOVL C00259 V=800.0 PL=0
MOVL C00260 V=800.0 PL=0
MOVL C00261 V=800.0 PL=0
MOVL C00262 V=800.0 PL=0
MOVL C00263 V=800.0 PL=0
MOVL C00264 V=800.0 PL=0
MOVL C00265 V=800.0 PL=0
MOVL C00266 V=800.0 PL=0
MOVL C00267 V=800.0 PL=0
MOVL C00268 V=800.0 PL=0
MOVL C00269 V=800.0 PL=0
MOVL C00270 V=800.0 PL=0
MOVL C00271 V=800.0 PL=0
MOVL C00272 V=800.0 PL=0
MOVL C00273 V=800.0 PL=0
MOVL C00274 V=800.0 PL=0
MOVL C00275 V=800.0 PL=0
MOVL C00276 V=800.0 PL=0
MOVL C00277 V=800.0 PL=0
MOVL C00278 V=800.0 PL=0
MOVL C00279 V=800.0 PL=0
MOVL C00280 V=800.0 PL=0
MOVL C00281 V=800.0 PL=0
MOVL C00282 V=800.0 PL=0
MOVL C00283 V=800.0 PL=0
MOVL C00284 V=800.0 PL=0
MOVL C00285 V=800.0 PL=0
MOVL C00286 V=800.0 PL=0
MOVL C00287 V=800.0 PL=0
MOVL C00288 V=800.0 PL=0
MOVL C00289 V=800.0 PL=0
MOVL C00290 V=800.0 PL=0
MOVL C00291 V=800.0 PL=0
MOVL C00292 V=800.0 PL=0
MOVL C00293 V=800.0 PL=0
MOVL C00294 V=800.0 PL=0
MOVL C00295 V=800.0 PL=0
MOVL C00296 V=800.0 PL=0
MOVL C00297 V=800.0 PL=0
MOVL C00298 V=800.0 PL=0
MOVL C00299 V=800.0 PL=0
MOVL C00300 V=800.0 PL=0
MOVL C00301 V=800.0 PL=0
MOVL C00302 V=800.0 PL=0
MOVL C00303 V=800.0 PL=0
MOVL C00304 V=800.0 PL=0
MOVL C00305 V=800.0 PL=0
MOVL C00306 V=800.0 PL=0
MOVL C00307 V=800.0 PL=0
MOVL C00308 V=800.0 PL=0
MOVL C00309 V=800.0 PL=0
MOVL C00310 V=800.0 PL=0
MOVL C00311 V=800.0 PL=0
MOVL C00312 V=800.0 PL=0
MOVL C00313 V=800.0 PL=0
MOVL C00314 V=800.0 PL=0
MOVL C00315 V=800.0 PL=0
MOVL C00316 V=800.0 PL=0
MOVL C00317 V=800.0 PL=0
MOVL C00318 V=800.0 PL=0
MOVL C00319 V=800.0 PL=0
MOVL C00320 V=800.0 PL=0
MOVL C00321 V=800.0 PL=0
MOVL C00322 V=800.0 PL=0
MOVL C00323 V=800.0 PL=0
MOVL C00324 V=800.0 PL=0
MOVL C00325 V=800.0 PL=0
MOVL C00326 V=800.0 PL=0
MOVL C00327 V=800.0 PL=0
MOVL C00328 V=800.0 PL=0
MOVL C00329 V=800.0 PL=0
MOVL C00330 V=800.0 PL=0
MOVL C00331 V=800.0 PL=0
MOVL C00332 V=800.0 PL=0
MOVL C00333 V=800.0 PL=0
MOVL C00334 V=800.0 PL=0
MOVL C00335 V=800.0 PL=0
MOVL C00336 V=800.0 PL=0
MOVL C00337 V=800.0 PL=0
MOVL C00338 V=800.0 PL=0
MOVL C00339 V=800.0 PL=0
MOVL C00340 V=800.0 PL=0
MOVL C00341 V=800.0 PL=0
MOVL C00342 V=800.0 PL=0
MOVL C00343 V=800.0 PL=0
MOVL C00344 V=800.0 PL=0
MOVL C00345 V=800.0 PL=0
MOVL C00346 V=800.0 PL=0
MOVL C00347 V=800.0 PL=0
MOVL C00348 V=800.0 PL=0
MOVL C00349 V=800.0 PL=0
MOVL C00350 V=800.0 PL=0
MOVL C00351 V=800.0 PL=0
MOVL C00352 V=800.0 PL=0
MOVL C00353 V=800.0 PL=0
MOVL C00354 V=800.0 PL=0
MOVL C00355 V=800.0 PL=0
MOVL C00356 V=800.0 PL=0
MOVL C00357 V=800.0 PL=0
MOVL C00358 V=800.0 PL=0
MOVL C00359 V=800.0 PL=0
MOVL C00360 V=800.0 PL=0
MOVL C00361 V=800.0 PL=0
MOVL C00362 V=800.0 PL=0
MOVL C00363 V=800.0 PL=0
MOVL C00364 V=800.0 PL=0
MOVL C00365 V=800.0 PL=0
MOVL C00366 V=800.0 PL=0
MOVL C00367 V=800.0 PL=0
MOVL C00368 V=800.0 PL=0
MOVL C00369 V=800.0 PL=0
MOVL C00370 V=800.0 PL=0
MOVL C00371 V=800.0 PL=0
MOVL C00372 V=800.0 PL=0
MOVL C00373 V=800.0 PL=0
MOVL C00374 V=800.0 PL=0
MOVL C00375 V=800.0 PL=0
MOVL C00376 V=800.0 PL=0
MOVL C00377 V=800.0 PL=0
MOVL C00378 V=800.0 PL=0
MOVL C00379 V=800.0 PL=0
MOVL C00380 V=800.0 PL=0
MOVL C00381 V=800.0 PL=0
MOVL C00382 V=800.0 PL=0
MOVL C00383 V=800.0 PL=0
MOVL C00384 V=800.0 PL=0
MOVL C00385 V=800.0 PL=0
MOVL C00386 V=800.0 PL=0
MOVL C00387 V=800.0 PL=0
MOVL C00388 V=800.0 PL=0
MOVL C00389 V=800.0 PL=0
MOVL C00390 V=800.0 PL=0
MOVL C00391 V=800.0 PL=0
MOVL C00392 V=800.0 PL=0
MOVL C00393 V=800.0 PL=0
MOVL C00394 V=800.0 PL=0
MOVL C00395 V=800.0 PL=0
MOVL C00396 V=800.0 PL=0
MOVL C00397 V=800.0 PL=0
MOVL C00398 V=800.0 PL=0
MOVL C00399 V=800.0 PL=0
MOVL C00400 V=800.0 PL=0
MOVL C00401 V=800.0 PL=0
MOVL C00402 V=800.0 PL=0
MOVL C00403 V=800.0 PL=0
MOVL C00404 V=800.0 PL=0
MOVL C00405 V=800.0 PL=0
MOVL C00406 V=800.0 PL=0
MOVL C00407 V=800.0 PL=0
MOVL C00408 V=800.0 PL=0
MOVL C00409 V=800.0 PL=0
MOVL C00410 V=800.0 PL=0
MOVL C00411 V=800.0 PL=0
MOVL C00412 V=800.0 PL=0
MOVL C00413 V=800.0 PL=0
MOVL C00414 V=800.0 PL=0
MOVL C00415 V=800.0 PL=0
MOVL C00416 V=800.0 PL=0
MOVL C00417 V=800.0 PL=0
MOVL C00418 V=800.0 PL=0
MOVL C00419 V=800.0 PL=0
MOVL C00420 V=800.0 PL=0
MOVL C00421 V=800.0 PL=0
MOVL C00422 V=800.0 PL=0
MOVL C00423 V=800.0 PL=0
MOVL C00424 V=800.0 PL=0
MOVL C00425 V=800.0 PL=0
MOVL C00426 V=800.0 PL=0
MOVL C00427 V=800.0 PL=0
MOVL C00428 V=800.0 PL=0
MOVL C00429 V=800.0 PL=0
MOVL C00430 V=800.0 PL=0
MOVL C00431 V=800.0 PL=0
MOVL C00432 V=800.0 PL=0
MOVL C00433 V=800.0 PL=0
MOVL C00434 V=800.0 PL=0
MOVL C00435 V=800.0 PL=0
MOVL C00436 V=800.0 PL=0
MOVL C00437 V=800.0 PL=0
MOVL C00438 V=800.0 PL=0
MOVL C00439 V=800.0 PL=0
MOVL C00440 V=800.0 PL=0
MOVL C00441 V=800.0 PL=0
MOVL C00442 V=800.0 PL=0
MOVL C00443 V=800.0 PL=0
MOVL C00444 V=800.0 PL=0
MOVL C00445 V=800.0 PL=0
MOVL C00446 V=800.0 PL=0
MOVL C00447 V=800.0 PL=0
MOVL C00448 V=800.0 PL=0
MOVL C00449 V=800.0 PL=0
MOVL C00450 V=800.0 PL=0
MOVL C00451 V=800.0 PL=0
MOVL C00452 V=800.0 PL=0
MOVL C00453 V=800.0 PL=0
MOVL C00454 V=800.0 PL=0
MOVL C00455 V=800.0 PL=0
MOVL C00456 V=800.0 PL=0
MOVL C00457 V=800.0 PL=0
MOVL C00458 V=800.0 PL=0
MOVL C00459 V=800.0 PL=0
MOVL C00460 V=800.0 PL=0
MOVL C00461 V=800.0 PL=0
MOVL C00462 V=800.0 PL=0
MOVL C00463 V=800.0 PL=0
MOVL C00464 V=800.0 PL=0
MOVL C00465 V=800.0 PL=0
MOVL C00466 V=800.0 PL=0
MOVL C00467 V=800.0 PL=0
MOVL C00468 V=800.0 PL=0
MOVL C00469 V=800.0 PL=0
MOVL C00470 V=800.0 PL=0
MOVL C00471 V=800.0 PL=0
MOVL C00472 V=800.0 PL=0
MOVL C00473 V=800.0 PL=0
MOVL C00474 V=800.0 PL=0
MOVL C00475 V=800.0 PL=0
MOVL C00476 V=800.0 PL=0
MOVL C00477 V=800.0 PL=0
MOVL C00478 V=800.0 PL=0
MOVL C00479 V=800.0 PL=0
MOVL C00480 V=800.0 PL=0
MOVL C00481 V=800.0 PL=0
MOVL C00482 V=800.0 PL=0
MOVL C00483 V=800.0 PL=0
MOVL C00484 V=800.0 PL=0
MOVL C00485 V=800.0 PL=0
MOVL C00486 V=800.0 PL=0
MOVL C00487 V=800.0 PL=0
MOVL C00488 V=800.0 PL=0
MOVL C00489 V=800.0 PL=0
MOVL C00490 V=800.0 PL=0
MOVL C00491 V=800.0 PL=0
MOVL C00492 V=800.0 PL=0
MOVL C00493 V=800.0 PL=0
MOVL C00494 V=800.0 PL=0
MOVL C00495 V=800.0 PL=0
MOVL C00496 V=800.0 PL=0
MOVL C00497 V=800.0 PL=0
MOVL C00498 V=800.0 PL=0
MOVL C00499 V=800.0 PL=0
MOVL C00500 V=800.0 PL=0
MOVL C00501 V=800.0 PL=0
MOVL C00502 V=800.0 PL=0
MOVL C00503 V=800.0 PL=0
MOVL C00504 V=800.0 PL=0
MOVL C00505 V=800.0 PL=0
MOVL C00506 V=800.0 PL=0
MOVL C00507 V=800.0 PL=0
MOVL C00508 V=800.0 PL=0
MOVL C00509 V=800.0 PL=0
MOVL C00510 V=800.0 PL=0
MOVL C00511 V=800.0 PL=0
MOVL C00512 V=800.0 PL=0
MOVL C00513 V=800.0 PL=0
MOVL C00514 V=800.0 PL=0
MOVL C00515 V=800.0 PL=0
MOVL C00516 V=800.0 PL=0
MOVL C00517 V=800.0 PL=0
MOVL C00518 V=800.0 PL=0
MOVL C00519 V=800.0 PL=0
MOVL C00520 V=800.0 PL=0
MOVL C00521 V=800.0 PL=0
MOVL C00522 V=800.0 PL=0
MOVL C00523 V=800.0 PL=0
MOVL C00524 V=800.0 PL=0
MOVL C00525 V=800.0 PL=0
MOVL C00526 V=800.0 PL=0
MOVL C00527 V=800.0 PL=0
MOVL C00528 V=800.0 PL=0
MOVL C00529 V=800.0 PL=0
MOVL C00530 V=800.0 PL=0
MOVL C00531 V=800.0 PL=0
MOVL C00532 V=800.0 PL=0
MOVL C00533 V=800.0 PL=0
MOVL C00534 V=800.0 PL=0
MOVL C00535 V=800.0 PL=0
MOVL C00536 V=800.0 PL=0
MOVL C00537 V=800.0 PL=0
MOVL C00538 V=800.0 PL=0
MOVL C00539 V=800.0 PL=0
MOVL C00540 V=800.0 PL=0
MOVL C00541 V=800.0 PL=0
MOVL C00542 V=800.0 PL=0
MOVL C00543 V=800.0 PL=0
MOVL C00544 V=800.0 PL=0
MOVL C00545 V=800.0 PL=0
MOVL C00546 V=800.0 PL=0
MOVL C00547 V=800.0 PL=0
MOVL C00548 V=800.0 PL=0
MOVL C00549 V=800.0 PL=0
MOVL C00550 V=800.0 PL=0
MOVL C00551 V=800.0 PL=0
MOVL C00552 V=800.0 PL=0
MOVL C00553 V=800.0 PL=0
MOVL C00554 V=800.0 PL=0
MOVL C00555 V=800.0 PL=0
MOVL C00556 V=800.0 PL=0
MOVL C00557 V=800.0 PL=0
MOVL C00558 V=800.0 PL=0
MOVL C00559 V=800.0 PL=0
MOVL C00560 V=800.0 PL=0
MOVL C00561 V=800.0 PL=0
MOVL C00562 V=800.0 PL=0
MOVL C00563 V=800.0 PL=0
MOVL C00564 V=800.0 PL=0
MOVL C00565 V=800.0 PL=0
MOVL C00566 V=800.0 PL=0
MOVL C00567 V=800.0 PL=0
MOVL C00568 V=800.0 PL=0
MOVL C00569 V=800.0 PL=0
MOVL C00570 V=800.0 PL=0
MOVL C00571 V=800.0 PL=0
MOVL C00572 V=800.0 PL=0
MOVL C00573 V=800.0 PL=0
MOVL C00574 V=800.0 PL=0
MOVL C00575 V=800.0 PL=0
MOVL C00576 V=800.0 PL=0
MOVL C00577 V=800.0 PL=0
MOVL C00578 V=800.0 PL=0
MOVL C00579 V=800.0 PL=0
MOVL C00580 V=800.0 PL=0
MOVL C00581 V=800.0 PL=0
MOVL C00582 V=800.0 PL=0
MOVL C00583 V=800.0 PL=0
MOVL C00584 V=800.0 PL=0
MOVL C00585 V=800.0 PL=0
MOVL C00586 V=800.0 PL=0
MOVL C00587 V=800.0 PL=0
MOVL C00588 V=800.0 PL=0
MOVL C00589 V=800.0 PL=0
MOVL C00590 V=800.0 PL=0
MOVL C00591 V=800.0 PL=0
MOVL C00592 V=800.0 PL=0
MOVL C00593 V=800.0 PL=0
MOVL C00594 V=800.0 PL=0
MOVL C00595 V=800.0 PL=0
MOVL C00596 V=800.0 PL=0
MOVL C00597 V=800.0 PL=0
MOVL C00598 V=800.0 PL=0
MOVL C00599 V=800.0 PL=0
MOVL C00600 V=800.0 PL=0
MOVL C00601 V=800.0 PL=0
MOVL C00602 V=800.0 PL=0
MOVL C00603 V=800.0 PL=0
MOVL C00604 V=800.0 PL=0
MOVL C00605 V=800.0 PL=0
MOVL C00606 V=800.0 PL=0
MOVL C00607 V=800.0 PL=0
MOVL C00608 V=800.0 PL=0
MOVL C00609 V=800.0 PL=0
MOVL C00610 V=800.0 PL=0
MOVL C00611 V=800.0 PL=0
MOVL C00612 V=800.0 PL=0
MOVL C00613 V=800.0 PL=0
MOVL C00614 V=800.0 PL=0
MOVL C00615 V=800.0 PL=0
MOVL C00616 V=800.0 PL=0
MOVL C00617 V=800.0 PL=0
MOVL C00618 V=800.0 PL=0
MOVL C00619 V=800.0 PL=0
MOVL C00620 V=800.0 PL=0
MOVL C00621 V=800.0 PL=0
MOVL C00622 V=800.0 PL=0
MOVL C00623 V=800.0 PL=0
MOVL C00624 V=800.0 PL=0
MOVL C00625 V=800.0 PL=0
MOVL C00626 V=800.0 PL=0
MOVL C00627 V=800.0 PL=0
MOVL C00628 V=800.0 PL=0
MOVL C00629 V=800.0 PL=0
MOVL C00630 V=800.0 PL=0
MOVL C00631 V=800.0 PL=0
MOVL C00632 V=800.0 PL=0
MOVL C00633 V=800.0 PL=0
MOVL C00634 V=800.0 PL=0
MOVL C00635 V=800.0 PL=0
MOVL C00636 V=800.0 PL=0
MOVL C00637 V=800.0 PL=0
MOVL C00638 V=800.0 PL=0
MOVL C00639 V=800.0 PL=0
MOVL C00640 V=800.0 PL=0
MOVL C00641 V=800.0 PL=0
MOVL C00642 V=800.0 PL=0
MOVL C00643 V=800.0 PL=0
MOVL C00644 V=800.0 PL=0
MOVL C00645 V=800.0 PL=0
MOVL C00646 V=800.0 PL=0
MOVL C00647 V=800.0 PL=0
MOVL C00648 V=800.0 PL=0
MOVL C00649 V=800.0 PL=0
MOVL C00650 V=800.0 PL=0
MOVL C00651 V=800.0 PL=0
MOVL C00652 V=800.0 PL=0
MOVL C00653 V=800.0 PL=0
MOVL C00654 V=800.0 PL=0
MOVL C00655 V=800.0 PL=0
MOVL C00656 V=800.0 PL=0
MOVL C00657 V=800.0 PL=0
MOVL C00658 V=800.0 PL=0
MOVL C00659 V=800.0 PL=0
MOVL C00660 V=800.0 PL=0
MOVL C00661 V=800.0 PL=0
MOVL C00662 V=800.0 PL=0
MOVL C00663 V=800.0 PL=0
MOVL C00664 V=800.0 PL=0
MOVL C00665 V=800.0 PL=0
MOVL C00666 V=800.0 PL=0
MOVL C00667 V=800.0 PL=0
MOVL C00668 V=800.0 PL=0
MOVL C00669 V=800.0 PL=0
MOVL C00670 V=800.0 PL=0
MOVL C00671 V=800.0 PL=0
MOVL C00672 V=800.0 PL=0
MOVL C00673 V=800.0 PL=0
MOVL C00674 V=800.0 PL=0
MOVL C00675 V=800.0 PL=0
MOVL C00676 V=800.0 PL=0
MOVL C00677 V=800.0 PL=0
MOVL C00678 V=800.0 PL=0
MOVL C00679 V=800.0 PL=0
MOVL C00680 V=800.0 PL=0
MOVL C00681 V=800.0 PL=0
MOVL C00682 V=800.0 PL=0
MOVL C00683 V=800.0 PL=0
MOVL C00684 V=800.0 PL=0
MOVL C00685 V=800.0 PL=0
MOVL C00686 V=800.0 PL=0
MOVL C00687 V=800.0 PL=0
MOVL C00688 V=800.0 PL=0
MOVL C00689 V=800.0 PL=0
MOVL C00690 V=800.0 PL=0
MOVL C00691 V=800.0 PL=0
MOVL C00692 V=800.0 PL=0
MOVL C00693 V=800.0 PL=0
MOVL C00694 V=800.0 PL=0
MOVL C00695 V=800.0 PL=0
MOVL C00696 V=800.0 PL=0
MOVL C00697 V=800.0 PL=0
MOVL C00698 V=800.0 PL=0
MOVL C00699 V=800.0 PL=0
MOVL C00700 V=800.0 PL=0
MOVL C00701 V=800.0 PL=0
MOVL C00702 V=800.0 PL=0
MOVL C00703 V=800.0 PL=0
MOVL C00704 V=800.0 PL=0
MOVL C00705 V=800.0 PL=0
MOVL C00706 V=800.0 PL=0
MOVL C00707 V=800.0 PL=0
MOVL C00708 V=800.0 PL=0
MOVL C00709 V=800.0 PL=0
MOVL C00710 V=800.0 PL=0
MOVL C00711 V=800.0 PL=0
MOVL C00712 V=800.0 PL=0
MOVL C00713 V=800.0 PL=0
MOVL C00714 V=800.0 PL=0
MOVL C00715 V=800.0 PL=0
MOVL C00716 V=800.0 PL=0
MOVL C00717 V=800.0 PL=0
MOVL C00718 V=800.0 PL=0
MOVL C00719 V=800.0 PL=0
MOVL C00720 V=800.0 PL=0
MOVL C00721 V=800.0 PL=0
MOVL C00722 V=800.0 PL=0
MOVL C00723 V=800.0 PL=0
MOVL C00724 V=800.0 PL=0
MOVL C00725 V=800.0 PL=0
MOVL C00726 V=800.0 PL=0
MOVL C00727 V=800.0 PL=0
MOVL C00728 V=800.0 PL=0
MOVL C00729 V=800.0 PL=0
MOVL C00730 V=800.0 PL=0
MOVL C00731 V=800.0 PL=0
MOVL C00732 V=800.0 PL=0
MOVL C00733 V=800.0 PL=0
MOVL C00734 V=800.0 PL=0
MOVL C00735 V=800.0 PL=0
MOVL C00736 V=800.0 PL=0
MOVL C00737 V=800.0 PL=0
MOVL C00738 V=800.0 PL=0
MOVL C00739 V=800.0 PL=0
MOVL C00740 V=800.0 PL=0
MOVL C00741 V=800.0 PL=0
MOVL C00742 V=800.0 PL=0
MOVL C00743 V=800.0 PL=0
MOVL C00744 V=800.0 PL=0
MOVL C00745 V=800.0 PL=0
MOVL C00746 V=800.0 PL=0
MOVL C00747 V=800.0 PL=0
MOVL C00748 V=800.0 PL=0
MOVL C00749 V=800.0 PL=0
MOVL C00750 V=800.0 PL=0
MOVL C00751 V=800.0 PL=0
MOVL C00752 V=800.0 PL=0
MOVL C00753 V=800.0 PL=0
MOVL C00754 V=800.0 PL=0
MOVL C00755 V=800.0 PL=0
MOVL C00756 V=800.0 PL=0
MOVL C00757 V=800.0 PL=0
MOVL C00758 V=800.0 PL=0
MOVL C00759 V=800.0 PL=0
MOVL C00760 V=800.0 PL=0
MOVL C00761 V=800.0 PL=0
MOVL C00762 V=800.0 PL=0
MOVL C00763 V=800.0 PL=0
MOVL C00764 V=800.0 PL=0
MOVL C00765 V=800.0 PL=0
MOVL C00766 V=800.0 PL=0
MOVL C00767 V=800.0 PL=0
MOVL C00768 V=800.0 PL=0
MOVL C00769 V=800.0 PL=0
MOVL C00770 V=800.0 PL=0
MOVL C00771 V=800.0 PL=0
MOVL C00772 V=800.0 PL=0
MOVL C00773 V=800.0 PL=0
MOVL C00774 V=800.0 PL=0
MOVL C00775 V=800.0 PL=0
MOVL C00776 V=800.0 PL=0
MOVL C00777 V=800.0 PL=0
MOVL C00778 V=800.0 PL=0
MOVL C00779 V=800.0 PL=0
MOVL C00780 V=800.0 PL=0
MOVL C00781 V=800.0 PL=0
MOVL C00782 V=800.0 PL=0
MOVL C00783 V=800.0 PL=0
MOVL C00784 V=800.0 PL=0
MOVL C00785 V=800.0 PL=0
MOVL C00786 V=800.0 PL=0
MOVL C00787 V=800.0 PL=0
MOVL C00788 V=800.0 PL=0
MOVL C00789 V=800.0 PL=0
MOVL C00790 V=800.0 PL=0
MOVL C00791 V=800.0 PL=0
MOVL C00792 V=800.0 PL=0
MOVL C00793 V=800.0 PL=0
MOVL C00794 V=800.0 PL=0
MOVL C00795 V=800.0 PL=0
MOVL C00796 V=800.0 PL=0
MOVL C00797 V=800.0 PL=0
MOVL C00798 V=800.0 PL=0
MOVL C00799 V=800.0 PL=0
MOVL C00800 V=800.0 PL=0
MOVL C00801 V=800.0 PL=0
MOVL C00802 V=800.0 PL=0
MOVL C00803 V=800.0 PL=0
MOVL C00804 V=800.0 PL=0
MOVL C00805 V=800.0 PL=0
MOVL C00806 V=800.0 PL=0
MOVL C00807 V=800.0 PL=0
MOVL C00808 V=800.0 PL=0
MOVL C00809 V=800.0 PL=0
MOVL C00810 V=800.0 PL=0
MOVL C00811 V=800.0 PL=0
MOVL C00812 V=800.0 PL=0
MOVL C00813 V=800.0 PL=0
MOVL C00814 V=800.0 PL=0
MOVL C00815 V=800.0 PL=0
MOVL C00816 V=800.0 PL=0
MOVL C00817 V=800.0 PL=0
MOVL C00818 V=800.0 PL=0
MOVL C00819 V=800.0 PL=0
MOVL C00820 V=800.0 PL=0
MOVL C00821 V=800.0 PL=0
MOVL C00822 V=800.0 PL=0
MOVL C00823 V=800.0 PL=0
MOVL C00824 V=800.0 PL=0
MOVL C00825 V=800.0 PL=0
MOVL C00826 V=800.0 PL=0
MOVL C00827 V=800.0 PL=0
MOVL C00828 V=800.0 PL=0
MOVL C00829 V=800.0 PL=0
MOVL C00830 V=800.0 PL=0
MOVL C00831 V=800.0 PL=0
MOVL C00832 V=800.0 PL=0
MOVL C00833 V=800.0 PL=0
MOVL C00834 V=800.0 PL=0
MOVL C00835 V=800.0 PL=0
MOVL C00836 V=800.0 PL=0
MOVL C00837 V=800.0 PL=0
MOVL C00838 V=800.0 PL=0
MOVL C00839 V=800.0 PL=0
MOVL C00840 V=800.0 PL=0
MOVL C00841 V=800.0 PL=0
MOVL C00842 V=800.0 PL=0
MOVL C00843 V=800.0 PL=0
MOVL C00844 V=800.0 PL=0
MOVL C00845 V=800.0 PL=0
MOVL C00846 V=800.0 PL=0
MOVL C00847 V=800.0 PL=0
MOVL C00848 V=800.0 PL=0
MOVL C00849 V=800.0 PL=0
MOVL C00850 V=800.0 PL=0
MOVL C00851 V=800.0 PL=0
MOVL C00852 V=800.0 PL=0
MOVL C00853 V=800.0 PL=0
MOVL C00854 V=800.0 PL=0
MOVL C00855 V=800.0 PL=0
MOVL C00856 V=800.0 PL=0
MOVL C00857 V=800.0 PL=0
MOVL C00858 V=800.0 PL=0
MOVL C00859 V=800.0 PL=0
MOVL C00860 V=800.0 PL=0
MOVL C00861 V=800.0 PL=0
MOVL C00862 V=800.0 PL=0
MOVL C00863 V=800.0 PL=0
MOVL C00864 V=800.0 PL=0
MOVL C00865 V=800.0 PL=0
MOVL C00866 V=800.0 PL=0
MOVL C00867 V=800.0 PL=0
MOVL C00868 V=800.0 PL=0
MOVL C00869 V=800.0 PL=0
MOVL C00870 V=800.0 PL=0
MOVL C00871 V=800.0 PL=0
MOVL C00872 V=800.0 PL=0
MOVL C00873 V=800.0 PL=0
MOVL C00874 V=800.0 PL=0
MOVL C00875 V=800.0 PL=0
MOVL C00876 V=800.0 PL=0
MOVL C00877 V=800.0 PL=0
MOVL C00878 V=800.0 PL=0
MOVL C00879 V=800.0 PL=0
MOVL C00880 V=800.0 PL=0
MOVL C00881 V=800.0 PL=0
MOVL C00882 V=800.0 PL=0
MOVL C00883 V=800.0 PL=0
MOVL C00884 V=800.0 PL=0
MOVL C00885 V=800.0 PL=0
MOVL C00886 V=800.0 PL=0
MOVL C00887 V=800.0 PL=0
MOVL C00888 V=800.0 PL=0
MOVL C00889 V=800.0 PL=0
MOVL C00890 V=800.0 PL=0
MOVL C00891 V=800.0 PL=0
MOVL C00892 V=800.0 PL=0
MOVL C00893 V=800.0 PL=0
MOVL C00894 V=800.0 PL=0
MOVL C00895 V=800.0 PL=0
MOVL C00896 V=800.0 PL=0
MOVL C00897 V=800.0 PL=0
MOVL C00898 V=800.0 PL=0
MOVL C00899 V=800.0 PL=0
MOVL C00900 V=800.0 PL=0
MOVL C00901 V=800.0 PL=0
MOVL C00902 V=800.0 PL=0
MOVL C00903 V=800.0 PL=0
MOVL C00904 V=800.0 PL=0
MOVL C00905 V=800.0 PL=0
MOVL C00906 V=800.0 PL=0
MOVL C00907 V=800.0 PL=0
MOVL C00908 V=800.0 PL=0
MOVL C00909 V=800.0 PL=0
MOVL C00910 V=800.0 PL=0
MOVL C00911 V=800.0 PL=0
MOVL C00912 V=800.0 PL=0
MOVL C00913 V=800.0 PL=0
MOVL C00914 V=800.0 PL=0
MOVL C00915 V=800.0 PL=0
MOVL C00916 V=800.0 PL=0
MOVL C00917 V=800.0 PL=0
MOVL C00918 V=800.0 PL=0
MOVL C00919 V=800.0 PL=0
MOVL C00920 V=800.0 PL=0
MOVL C00921 V=800.0 PL=0
MOVL C00922 V=800.0 PL=0
MOVL C00923 V=800.0 PL=0
MOVL C00924 V=800.0 PL=0
MOVL C00925 V=800.0 PL=0
MOVL C00926 V=800.0 PL=0
MOVL C00927 V=800.0 PL=0
MOVL C00928 V=800.0 PL=0
MOVL C00929 V=800.0 PL=0
MOVL C00930 V=800.0 PL=0
MOVL C00931 V=800.0 PL=0
MOVL C00932 V=800.0 PL=0
MOVL C00933 V=800.0 PL=0
MOVL C00934 V=800.0 PL=0
MOVL C00935 V=800.0 PL=0
MOVL C00936 V=800.0 PL=0
MOVL C00937 V=800.0 PL=0
MOVL C00938 V=800.0 PL=0
MOVL C00939 V=800.0 PL=0
MOVL C00940 V=800.0 PL=0
MOVL C00941 V=800.0 PL=0
MOVL C00942 V=800.0 PL=0
MOVL C00943 V=800.0 PL=0
MOVL C00944 V=800.0 PL=0
MOVL C00945 V=800.0 PL=0
MOVL C00946 V=800.0 PL=0
MOVL C00947 V=800.0 PL=0
MOVL C00948 V=800.0 PL=0
MOVL C00949 V=800.0 PL=0
MOVL C00950 V=800.0 PL=0
MOVL C00951 V=800.0 PL=0
MOVL C00952 V=800.0 PL=0
MOVL C00953 V=800.0 PL=0
MOVL C00954 V=800.0 PL=0
MOVL C00955 V=800.0 PL=0
MOVL C00956 V=800.0 PL=0
MOVL C00957 V=800.0 PL=0
MOVL C00958 V=800.0 PL=0
MOVL C00959 V=800.0 PL=0
MOVL C00960 V=800.0 PL=0
MOVL C00961 V=800.0 PL=0
MOVL C00962 V=800.0 PL=0
MOVL C00963 V=800.0 PL=0
MOVL C00964 V=800.0 PL=0
MOVL C00965 V=800.0 PL=0
MOVL C00966 V=800.0 PL=0
MOVL C00967 V=800.0 PL=0
MOVL C00968 V=800.0 PL=0
MOVL C00969 V=800.0 PL=0
MOVL C00970 V=800.0 PL=0
MOVL C00971 V=800.0 PL=0
MOVL C00972 V=800.0 PL=0
MOVL C00973 V=800.0 PL=0
MOVL C00974 V=800.0 PL=0
MOVL C00975 V=800.0 PL=0
MOVL C00976 V=800.0 PL=0
MOVL C00977 V=800.0 PL=0
MOVL C00978 V=800.0 PL=0
MOVL C00979 V=800.0 PL=0
MOVL C00980 V=800.0 PL=0
MOVL C00981 V=800.0 PL=0
MOVL C00982 V=800.0 PL=0
MOVL C00983 V=800.0 PL=0
MOVL C00984 V=800.0 PL=0
MOVL C00985 V=800.0 PL=0
MOVL C00986 V=800.0 PL=0
MOVL C00987 V=800.0 PL=0
MOVL C00988 V=800.0 PL=0
MOVL C00989 V=800.0 PL=0
MOVL C00990 V=800.0 PL=0
MOVL C00991 V=800.0 PL=0
MOVL C00992 V=800.0 PL=0
MOVL C00993 V=800.0 PL=0
MOVL C00994 V=800.0 PL=0
MOVL C00995 V=800.0 PL=0
MOVL C00996 V=800.0 PL=0
MOVL C00997 V=800.0 PL=0
MOVL C00998 V=800.0 PL=0
MOVL C00999 V=800.0 PL=0
MOVL C01000 V=800.0 PL=0
MOVL C01001 V=800.0 PL=0
MOVL C01002 V=800.0 PL=0
MOVL C01003 V=800.0 PL=0
MOVL C01004 V=800.0 PL=0
MOVL C01005 V=800.0 PL=0
MOVL C01006 V=800.0 PL=0
MOVL C01007 V=800.0 PL=0
MOVL C01008 V=800.0 PL=0
MOVL C01009 V=800.0 PL=0
MOVL C01010 V=800.0 PL=0
MOVL C01011 V=800.0 PL=0
MOVL C01012 V=800.0 PL=0
MOVL C01013 V=800.0 PL=0
MOVL C01014 V=800.0 PL=0
MOVL C01015 V=800.0 PL=0
MOVL C01016 V=800.0 PL=0
MOVL C01017 V=800.0 PL=0
MOVL C01018 V=800.0 PL=0
MOVL C01019 V=800.0 PL=0
MOVL C01020 V=800.0 PL=0
MOVL C01021 V=800.0 PL=0
MOVL C01022 V=800.0 PL=0
MOVL C01023 V=800.0 PL=0
MOVL C01024 V=800.0 PL=0
MOVL C01025 V=800.0 PL=0
MOVL C01026 V=800.0 PL=0
MOVL C01027 V=800.0 PL=0
MOVL C01028 V=800.0 PL=0
MOVL C01029 V=800.0 PL=0
MOVL C01030 V=800.0 PL=0
MOVL C01031 V=800.0 PL=0
MOVL C01032 V=800.0 PL=0
MOVL C01033 V=800.0 PL=0
MOVL C01034 V=800.0 PL=0
MOVL C01035 V=800.0 PL=0
MOVL C01036 V=800.0 PL=0
MOVL C01037 V=800.0 PL=0
MOVL C01038 V=800.0 PL=0
MOVL C01039 V=800.0 PL=0
MOVL C01040 V=800.0 PL=0
MOVL C01041 V=800.0 PL=0
MOVL C01042 V=800.0 PL=0
MOVL C01043 V=800.0 PL=0
MOVL C01044 V=800.0 PL=0
MOVL C01045 V=800.0 PL=0
MOVL C01046 V=800.0 PL=0
MOVL C01047 V=800.0 PL=0
MOVL C01048 V=800.0 PL=0
MOVL C01049 V=800.0 PL=0
MOVL C01050 V=800.0 PL=0
MOVL C01051 V=800.0 PL=0
MOVL C01052 V=800.0 PL=0
MOVL C01053 V=800.0 PL=0
MOVL C01054 V=800.0 PL=0
MOVL C01055 V=800.0 PL=0
MOVL C01056 V=800.0 PL=0
MOVL C01057 V=800.0 PL=0
MOVL C01058 V=800.0 PL=0
MOVL C01059 V=800.0 PL=0
MOVL C01060 V=800.0 PL=0
MOVL C01061 V=800.0 PL=0
MOVL C01062 V=800.0 PL=0
MOVL C01063 V=800.0 PL=0
MOVL C01064 V=800.0 PL=0
MOVL C01065 V=800.0 PL=0
MOVL C01066 V=800.0 PL=0
MOVL C01067 V=800.0 PL=0
MOVL C01068 V=800.0 PL=0
MOVL C01069 V=800.0 PL=0
MOVL C01070 V=800.0 PL=0
MOVL C01071 V=800.0 PL=0
MOVL C01072 V=800.0 PL=0
MOVL C01073 V=800.0 PL=0
MOVL C01074 V=800.0 PL=0
MOVL C01075 V=800.0 PL=0
MOVL C01076 V=800.0 PL=0
MOVL C01077 V=800.0 PL=0
MOVL C01078 V=800.0 PL=0
MOVL C01079 V=800.0 PL=0
MOVL C01080 V=800.0 PL=0
MOVL C01081 V=800.0 PL=0
MOVL C01082 V=800.0 PL=0
MOVL C01083 V=800.0 PL=0
MOVL C01084 V=800.0 PL=0
MOVL C01085 V=800.0 PL=0
MOVL C01086 V=800.0 PL=0
MOVL C01087 V=800.0 PL=0
MOVL C01088 V=800.0 PL=0
MOVL C01089 V=800.0 PL=0
MOVL C01090 V=800.0 PL=0
MOVL C01091 V=800.0 PL=0
MOVL C01092 V=800.0 PL=0
MOVL C01093 V=800.0 PL=0
MOVL C01094 V=800.0 PL=0
MOVL C01095 V=800.0 PL=0
MOVL C01096 V=800.0 PL=0
MOVL C01097 V=800.0 PL=0
MOVL C01098 V=800.0 PL=0
MOVL C01099 V=800.0 PL=0
MOVL C01100 V=800.0 PL=0
MOVL C01101 V=800.0 PL=0
MOVL C01102 V=800.0 PL=0
MOVL C01103 V=800.0 PL=0
MOVL C01104 V=800.0 PL=0
MOVL C01105 V=800.0 PL=0
MOVL C01106 V=800.0 PL=0
MOVL C01107 V=800.0 PL=0
MOVL C01108 V=800.0 PL=0
MOVL C01109 V=800.0 PL=0
MOVL C01110 V=800.0 PL=0
MOVL C01111 V=800.0 PL=0
MOVL C01112 V=800.0 PL=0
MOVL C01113 V=800.0 PL=0
MOVL C01114 V=800.0 PL=0
MOVL C01115 V=800.0 PL=0
MOVL C01116 V=800.0 PL=0
MOVL C01117 V=800.0 PL=0
MOVL C01118 V=800.0 PL=0
MOVL C01119 V=800.0 PL=0
MOVL C01120 V=800.0 PL=0
MOVL C01121 V=800.0 PL=0
MOVL C01122 V=800.0 PL=0
MOVL C01123 V=800.0 PL=0
MOVL C01124 V=800.0 PL=0
MOVL C01125 V=800.0 PL=0
MOVL C01126 V=800.0 PL=0
MOVL C01127 V=800.0 PL=0
MOVL C01128 V=800.0 PL=0
MOVL C01129 V=800.0 PL=0
MOVL C01130 V=800.0 PL=0
MOVL C01131 V=800.0 PL=0
MOVL C01132 V=800.0 PL=0
MOVL C01133 V=800.0 PL=0
MOVL C01134 V=800.0 PL=0
MOVL C01135 V=800.0 PL=0
MOVL C01136 V=800.0 PL=0
MOVL C01137 V=800.0 PL=0
MOVL C01138 V=800.0 PL=0
MOVL C01139 V=800.0 PL=0
MOVL C01140 V=800.0 PL=0
MOVL C01141 V=800.0 PL=0
MOVL C01142 V=800.0 PL=0
MOVL C01143 V=800.0 PL=0
MOVL C01144 V=800.0 PL=0
MOVL C01145 V=800.0 PL=0
MOVL C01146 V=800.0 PL=0
MOVL C01147 V=800.0 PL=0
MOVL C01148 V=800.0 PL=0
MOVL C01149 V=800.0 PL=0
MOVL C01150 V=800.0 PL=0
MOVL C01151 V=800.0 PL=0
MOVL C01152 V=800.0 PL=0
MOVL C01153 V=800.0 PL=0
MOVL C01154 V=800.0 PL=0
MOVL C01155 V=800.0 PL=0
MOVL C01156 V=800.0 PL=0
MOVL C01157 V=800.0 PL=0
MOVL C01158 V=800.0 PL=0
MOVL C01159 V=800.0 PL=0
MOVL C01160 V=800.0 PL=0
MOVL C01161 V=800.0 PL=0
MOVL C01162 V=800.0 PL=0
MOVL C01163 V=800.0 PL=0
MOVL C01164 V=800.0 PL=0
MOVL C01165 V=800.0 PL=0
MOVL C01166 V=800.0 PL=0
MOVL C01167 V=800.0 PL=0
MOVL C01168 V=800.0 PL=0
MOVL C01169 V=800.0 PL=0
MOVL C01170 V=800.0 PL=0
MOVL C01171 V=800.0 PL=0
MOVL C01172 V=800.0 PL=0
MOVL C01173 V=800.0 PL=0
MOVL C01174 V=800.0 PL=0
MOVL C01175 V=800.0 PL=0
MOVL C01176 V=800.0 PL=0
MOVL C01177 V=800.0 PL=0
MOVL C01178 V=800.0 PL=0
MOVL C01179 V=800.0 PL=0
MOVL C01180 V=800.0 PL=0
MOVL C01181 V=800.0 PL=0
MOVL C01182 V=800.0 PL=0
MOVL C01183 V=800.0 PL=0
MOVL C01184 V=800.0 PL=0
MOVL C01185 V=800.0 PL=0
MOVL C01186 V=800.0 PL=0
MOVL C01187 V=800.0 PL=0
MOVL C01188 V=800.0 PL=0
MOVL C01189 V=800.0 PL=0
MOVL C01190 V=800.0 PL=0
MOVL C01191 V=800.0 PL=0
MOVL C01192 V=800.0 PL=0
MOVL C01193 V=800.0 PL=0
MOVL C01194 V=800.0 PL=0
MOVL C01195 V=800.0 PL=0
MOVL C01196 V=800.0 PL=0
MOVL C01197 V=800.0 PL=0
MOVL C01198 V=800.0 PL=0
MOVL C01199 V=800.0 PL=0
MOVL C01200 V=800.0 PL=0
MOVL C01201 V=800.0 PL=0
MOVL C01202 V=800.0 PL=0
MOVL C01203 V=800.0 PL=0
MOVL C01204 V=800.0 PL=0
MOVL C01205 V=800.0 PL=0
MOVL C01206 V=800.0 PL=0
MOVL C01207 V=800.0 PL=0
MOVL C01208 V=800.0 PL=0
MOVL C01209 V=800.0 PL=0
MOVL C01210 V=800.0 PL=0
MOVL C01211 V=800.0 PL=0
MOVL C01212 V=800.0 PL=0
MOVL C01213 V=800.0 PL=0
MOVL C01214 V=800.0 PL=0
MOVL C01215 V=800.0 PL=0
MOVL C01216 V=800.0 PL=0
MOVL C01217 V=800.0 PL=0
MOVL C01218 V=800.0 PL=0
MOVL C01219 V=800.0 PL=0
MOVL C01220 V=800.0 PL=0
MOVL C01221 V=800.0 PL=0
MOVL C01222 V=800.0 PL=0
MOVL C01223 V=800.0 PL=0
MOVL C01224 V=800.0 PL=0
MOVL C01225 V=800.0 PL=0
MOVL C01226 V=800.0 PL=0
MOVL C01227 V=800.0 PL=0
MOVL C01228 V=800.0 PL=0
MOVL C01229 V=800.0 PL=0
MOVL C01230 V=800.0 PL=0
MOVL C01231 V=800.0 PL=0
MOVL C01232 V=800.0 PL=0
MOVL C01233 V=800.0 PL=0
MOVL C01234 V=800.0 PL=0
MOVL C01235 V=800.0 PL=0
MOVL C01236 V=800.0 PL=0
MOVL C01237 V=800.0 PL=0
MOVL C01238 V=800.0 PL=0
MOVL C01239 V=800.0 PL=0
MOVL C01240 V=800.0 PL=0
MOVL C01241 V=800.0 PL=0
MOVL C01242 V=800.0 PL=0
MOVL C01243 V=800.0 PL=0
MOVL C01244 V=800.0 PL=0
MOVL C01245 V=800.0 PL=0
MOVL C01246 V=800.0 PL=0
MOVL C01247 V=800.0 PL=0
MOVL C01248 V=800.0 PL=0
MOVL C01249 V=800.0 PL=0
MOVL C01250 V=800.0 PL=0
MOVL C01251 V=800.0 PL=0
MOVL C01252 V=800.0 PL=0
MOVL C01253 V=800.0 PL=0
MOVL C01254 V=800.0 PL=0
MOVL C01255 V=800.0 PL=0
MOVL C01256 V=800.0 PL=0
MOVL C01257 V=800.0 PL=0
MOVL C01258 V=800.0 PL=0
MOVL C01259 V=800.0 PL=0
MOVL C01260 V=800.0 PL=0
MOVL C01261 V=800.0 PL=0
MOVL C01262 V=800.0 PL=0
MOVL C01263 V=800.0 PL=0
MOVL C01264 V=800.0 PL=0
MOVL C01265 V=800.0 PL=0
MOVL C01266 V=800.0 PL=0
MOVL C01267 V=800.0 PL=0
MOVL C01268 V=800.0 PL=0
MOVL C01269 V=800.0 PL=0
MOVL C01270 V=800.0 PL=0
MOVL C01271 V=800.0 PL=0
MOVL C01272 V=800.0 PL=0
MOVL C01273 V=800.0 PL=0
MOVL C01274 V=800.0 PL=0
MOVL C01275 V=800.0 PL=0
MOVL C01276 V=800.0 PL=0
MOVL C01277 V=800.0 PL=0
MOVL C01278 V=800.0 PL=0
MOVL C01279 V=800.0 PL=0
MOVL C01280 V=800.0 PL=0
MOVL C01281 V=800.0 PL=0
MOVL C01282 V=800.0 PL=0
MOVL C01283 V=800.0 PL=0
MOVL C01284 V=800.0 PL=0
MOVL C01285 V=800.0 PL=0
MOVL C01286 V=800.0 PL=0
MOVL C01287 V=800.0 PL=0
MOVL C01288 V=800.0 PL=0
MOVL C01289 V=800.0 PL=0
MOVL C01290 V=800.0 PL=0
MOVL C01291 V=800.0 PL=0
MOVL C01292 V=800.0 PL=0
MOVL C01293 V=800.0 PL=0
MOVL C01294 V=800.0 PL=0
MOVL C01295 V=800.0 PL=0
MOVL C01296 V=800.0 PL=0
MOVL C01297 V=800.0 PL=0
MOVL C01298 V=800.0 PL=0
MOVL C01299 V=800.0 PL=0
MOVL C01300 V=800.0 PL=0
MOVL C01301 V=800.0 PL=0
MOVL C01302 V=800.0 PL=0
MOVL C01303 V=800.0 PL=0
MOVL C01304 V=800.0 PL=0
MOVL C01305 V=800.0 PL=0
MOVL C01306 V=800.0 PL=0
MOVL C01307 V=800.0 PL=0
MOVL C01308 V=800.0 PL=0
MOVL C01309 V=800.0 PL=0
MOVL C01310 V=800.0 PL=0
MOVL C01311 V=800.0 PL=0
MOVL C01312 V=800.0 PL=0
MOVL C01313 V=800.0 PL=0
MOVL C01314 V=800.0 PL=0
MOVL C01315 V=800.0 PL=0
MOVL C01316 V=800.0 PL=0
MOVL C01317 V=800.0 PL=0
MOVL C01318 V=800.0 PL=0
MOVL C01319 V=800.0 PL=0
MOVL C01320 V=800.0 PL=0
MOVL C01321 V=800.0 PL=0
MOVL C01322 V=800.0 PL=0
MOVL C01323 V=800.0 PL=0
MOVL C01324 V=800.0 PL=0
MOVL C01325 V=800.0 PL=0
MOVL C01326 V=800.0 PL=0
MOVL C01327 V=800.0 PL=0
MOVL C01328 V=800.0 PL=0
MOVL C01329 V=800.0 PL=0
MOVL C01330 V=800.0 PL=0
MOVL C01331 V=800.0 PL=0
MOVL C01332 V=800.0 PL=0
MOVL C01333 V=800.0 PL=0
MOVL C01334 V=800.0 PL=0
MOVL C01335 V=800.0 PL=0
MOVL C01336 V=800.0 PL=0
MOVL C01337 V=800.0 PL=0
MOVL C01338 V=800.0 PL=0
MOVL C01339 V=800.0 PL=0
MOVL C01340 V=800.0 PL=0
MOVL C01341 V=800.0 PL=0
MOVL C01342 V=800.0 PL=0
MOVL C01343 V=800.0 PL=0
MOVL C01344 V=800.0 PL=0
MOVL C01345 V=800.0 PL=0
MOVL C01346 V=800.0 PL=0
MOVL C01347 V=800.0 PL=0
MOVL C01348 V=800.0 PL=0
MOVL C01349 V=800.0 PL=0
MOVL C01350 V=800.0 PL=0
MOVL C01351 V=800.0 PL=0
MOVL C01352 V=800.0 PL=0
MOVL C01353 V=800.0 PL=0
MOVL C01354 V=800.0 PL=0
MOVL C01355 V=800.0 PL=0
MOVL C01356 V=800.0 PL=0
MOVL C01357 V=800.0 PL=0
MOVL C01358 V=800.0 PL=0
MOVL C01359 V=800.0 PL=0
MOVL C01360 V=800.0 PL=0
MOVL C01361 V=800.0 PL=0
MOVL C01362 V=800.0 PL=0
MOVL C01363 V=800.0 PL=0
MOVL C01364 V=800.0 PL=0
MOVL C01365 V=800.0 PL=0
MOVL C01366 V=800.0 PL=0
MOVL C01367 V=800.0 PL=0
MOVL C01368 V=800.0 PL=0
MOVL C01369 V=800.0 PL=0
MOVL C01370 V=800.0 PL=0
MOVL C01371 V=800.0 PL=0
MOVL C01372 V=800.0 PL=0
MOVL C01373 V=800.0 PL=0
MOVL C01374 V=800.0 PL=0
MOVL C01375 V=800.0 PL=0
MOVL C01376 V=800.0 PL=0
MOVL C01377 V=800.0 PL=0
MOVL C01378 V=800.0 PL=0
MOVL C01379 V=800.0 PL=0
MOVL C01380 V=800.0 PL=0
MOVL C01381 V=800.0 PL=0
MOVL C01382 V=800.0 PL=0
MOVL C01383 V=800.0 PL=0
MOVL C01384 V=800.0 PL=0
MOVL C01385 V=800.0 PL=0
MOVL C01386 V=800.0 PL=0
MOVL C01387 V=800.0 PL=0
MOVL C01388 V=800.0 PL=0
MOVL C01389 V=800.0 PL=0
MOVL C01390 V=800.0 PL=0
MOVL C01391 V=800.0 PL=0
MOVL C01392 V=800.0 PL=0
MOVL C01393 V=800.0 PL=0
MOVL C01394 V=800.0 PL=0
MOVL C01395 V=800.0 PL=0
MOVL C01396 V=800.0 PL=0
MOVL C01397 V=800.0 PL=0
MOVL C01398 V=800.0 PL=0
MOVL C01399 V=800.0 PL=0
MOVL C01400 V=800.0 PL=0
MOVL C01401 V=800.0 PL=0
MOVL C01402 V=800.0 PL=0
MOVL C01403 V=800.0 PL=0
MOVL C01404 V=800.0 PL=0
MOVL C01405 V=800.0 PL=0
MOVL C01406 V=800.0 PL=0
MOVL C01407 V=800.0 PL=0
MOVL C01408 V=800.0 PL=0
MOVL C01409 V=800.0 PL=0
MOVL C01410 V=800.0 PL=0
MOVL C01411 V=800.0 PL=0
MOVL C01412 V=800.0 PL=0
MOVL C01413 V=800.0 PL=0
MOVL C01414 V=800.0 PL=0
MOVL C01415 V=800.0 PL=0
MOVL C01416 V=800.0 PL=0
MOVL C01417 V=800.0 PL=0
MOVL C01418 V=800.0 PL=0
MOVL C01419 V=800.0 PL=0
MOVL C01420 V=800.0 PL=0
MOVL C01421 V=800.0 PL=0
MOVL C01422 V=800.0 PL=0
MOVL C01423 V=800.0 PL=0
MOVL C01424 V=800.0 PL=0
MOVL C01425 V=800.0 PL=0
MOVL C01426 V=800.0 PL=0
MOVL C01427 V=800.0 PL=0
MOVL C01428 V=800.0 PL=0
MOVL C01429 V=800.0 PL=0
MOVL C01430 V=800.0 PL=0
MOVL C01431 V=800.0 PL=0
MOVL C01432 V=800.0 PL=0
MOVL C01433 V=800.0 PL=0
MOVL C01434 V=800.0 PL=0
MOVL C01435 V=800.0 PL=0
MOVL C01436 V=800.0 PL=0
MOVL C01437 V=800.0 PL=0
MOVL C01438 V=800.0 PL=0
MOVL C01439 V=800.0 PL=0
MOVL C01440 V=800.0 PL=0
MOVL C01441 V=800.0 PL=0
MOVL C01442 V=800.0 PL=0
MOVL C01443 V=800.0 PL=0
MOVL C01444 V=800.0 PL=0
MOVL C01445 V=800.0 PL=0
MOVL C01446 V=800.0 PL=0
MOVL C01447 V=800.0 PL=0
MOVL C01448 V=800.0 PL=0
MOVL C01449 V=800.0 PL=0
MOVL C01450 V=800.0 PL=0
MOVL C01451 V=800.0 PL=0
MOVL C01452 V=800.0 PL=0
MOVL C01453 V=800.0 PL=0
MOVL C01454 V=800.0 PL=0
MOVL C01455 V=800.0 PL=0
MOVL C01456 V=800.0 PL=0
MOVL C01457 V=800.0 PL=0
MOVL C01458 V=800.0 PL=0
MOVL C01459 V=800.0 PL=0
MOVL C01460 V=800.0 PL=0
MOVL C01461 V=800.0 PL=0
MOVL C01462 V=800.0 PL=0
MOVL C01463 V=800.0 PL=0
MOVL C01464 V=800.0 PL=0
MOVL C01465 V=800.0 PL=0
MOVL C01466 V=800.0 PL=0
MOVL C01467 V=800.0 PL=0
MOVL C01468 V=800.0 PL=0
MOVL C01469 V=800.0 PL=0
MOVL C01470 V=800.0 PL=0
MOVL C01471 V=800.0 PL=0
MOVL C01472 V=800.0 PL=0
MOVL C01473 V=800.0 PL=0
MOVL C01474 V=800.0 PL=0
MOVL C01475 V=800.0 PL=0
MOVL C01476 V=800.0 PL=0
MOVL C01477 V=800.0 PL=0
MOVL C01478 V=800.0 PL=0
MOVL C01479 V=800.0 PL=0
MOVL C01480 V=800.0 PL=0
MOVL C01481 V=800.0 PL=0
MOVL C01482 V=800.0 PL=0
MOVL C01483 V=800.0 PL=0
MOVL C01484 V=800.0 PL=0
MOVL C01485 V=800.0 PL=0
MOVL C01486 V=800.0 PL=0
MOVL C01487 V=800.0 PL=0
MOVL C01488 V=800.0 PL=0
MOVL C01489 V=800.0 PL=0
MOVL C01490 V=800.0 PL=0
MOVL C01491 V=800.0 PL=0
MOVL C01492 V=800.0 PL=0
MOVL C01493 V=800.0 PL=0
MOVL C01494 V=800.0 PL=0
MOVL C01495 V=800.0 PL=0
MOVL C01496 V=800.0 PL=0
MOVL C01497 V=800.0 PL=0
MOVL C01498 V=800.0 PL=0
MOVL C01499 V=800.0 PL=0
MOVL C01500 V=800.0 PL=0
MOVL C01501 V=800.0 PL=0
MOVL C01502 V=800.0 PL=0
MOVL C01503 V=800.0 PL=0
MOVL C01504 V=800.0 PL=0
MOVL C01505 V=800.0 PL=0
MOVL C01506 V=800.0 PL=0
MOVL C01507 V=800.0 PL=0
MOVL C01508 V=800.0 PL=0
MOVL C01509 V=800.0 PL=0
MOVL C01510 V=800.0 PL=0
MOVL C01511 V=800.0 PL=0
MOVL C01512 V=800.0 PL=0
MOVL C01513 V=800.0 PL=0
MOVL C01514 V=800.0 PL=0
MOVL C01515 V=800.0 PL=0
MOVL C01516 V=800.0 PL=0
MOVL C01517 V=800.0 PL=0
MOVL C01518 V=800.0 PL=0
MOVL C01519 V=800.0 PL=0
MOVL C01520 V=800.0 PL=0
MOVL C01521 V=800.0 PL=0
MOVL C01522 V=800.0 PL=0
MOVL C01523 V=800.0 PL=0
MOVL C01524 V=800.0 PL=0
MOVL C01525 V=800.0 PL=0
MOVL C01526 V=800.0 PL=0
MOVL C01527 V=800.0 PL=0
MOVL C01528 V=800.0 PL=0
MOVL C01529 V=800.0 PL=0
MOVL C01530 V=800.0 PL=0
MOVL C01531 V=800.0 PL=0
MOVL C01532 V=800.0 PL=0
MOVL C01533 V=800.0 PL=0
MOVL C01534 V=800.0 PL=0
MOVL C01535 V=800.0 PL=0
MOVL C01536 V=800.0 PL=0
MOVL C01537 V=800.0 PL=0
MOVL C01538 V=800.0 PL=0
MOVL C01539 V=800.0 PL=0
MOVL C01540 V=800.0 PL=0
MOVL C01541 V=800.0 PL=0
MOVL C01542 V=800.0 PL=0
MOVL C01543 V=800.0 PL=0
MOVL C01544 V=800.0 PL=0
MOVL C01545 V=800.0 PL=0
MOVL C01546 V=800.0 PL=0
MOVL C01547 V=800.0 PL=0
MOVL C01548 V=800.0 PL=0
MOVL C01549 V=800.0 PL=0
MOVL C01550 V=800.0 PL=0
MOVL C01551 V=800.0 PL=0
MOVL C01552 V=800.0 PL=0
MOVL C01553 V=800.0 PL=0
MOVL C01554 V=800.0 PL=0
MOVL C01555 V=800.0 PL=0
MOVL C01556 V=800.0 PL=0
MOVL C01557 V=800.0 PL=0
MOVL C01558 V=800.0 PL=0
MOVL C01559 V=800.0 PL=0
MOVL C01560 V=800.0 PL=0
MOVL C01561 V=800.0 PL=0
MOVL C01562 V=800.0 PL=0
MOVL C01563 V=800.0 PL=0
MOVL C01564 V=800.0 PL=0
MOVL C01565 V=800.0 PL=0
MOVL C01566 V=800.0 PL=0
MOVL C01567 V=800.0 PL=0
MOVL C01568 V=800.0 PL=0
MOVL C01569 V=800.0 PL=0
MOVL C01570 V=800.0 PL=0
MOVL C01571 V=800.0 PL=0
MOVL C01572 V=800.0 PL=0
MOVL C01573 V=800.0 PL=0
MOVL C01574 V=800.0 PL=0
MOVL C01575 V=800.0 PL=0
MOVL C01576 V=800.0 PL=0
MOVL C01577 V=800.0 PL=0
MOVL C01578 V=800.0 PL=0
MOVL C01579 V=800.0 PL=0
MOVL C01580 V=800.0 PL=0
MOVL C01581 V=800.0 PL=0
MOVL C01582 V=800.0 PL=0
MOVL C01583 V=800.0 PL=0
MOVL C01584 V=800.0 PL=0
MOVL C01585 V=800.0 PL=0
MOVL C01586 V=800.0 PL=0
MOVL C01587 V=800.0 PL=0
MOVL C01588 V=800.0 PL=0
MOVL C01589 V=800.0 PL=0
MOVL C01590 V=800.0 PL=0
MOVL C01591 V=800.0 PL=0
MOVL C01592 V=800.0 PL=0
MOVL C01593 V=800.0 PL=0
MOVL C01594 V=800.0 PL=0
MOVL C01595 V=800.0 PL=0
MOVL C01596 V=800.0 PL=0
MOVL C01597 V=800.0 PL=0
MOVL C01598 V=800.0 PL=0
MOVL C01599 V=800.0 PL=0
MOVL C01600 V=800.0 PL=0
MOVL C01601 V=800.0 PL=0
MOVL C01602 V=800.0 PL=0
MOVL C01603 V=800.0 PL=0
MOVL C01604 V=800.0 PL=0
MOVL C01605 V=800.0 PL=0
MOVL C01606 V=800.0 PL=0
MOVL C01607 V=800.0 PL=0
MOVL C01608 V=800.0 PL=0
MOVL C01609 V=800.0 PL=0
MOVL C01610 V=800.0 PL=0
MOVL C01611 V=800.0 PL=0
MOVL C01612 V=800.0 PL=0
MOVL C01613 V=800.0 PL=0
MOVL C01614 V=800.0 PL=0
MOVL C01615 V=800.0 PL=0
MOVL C01616 V=800.0 PL=0
MOVL C01617 V=800.0 PL=0
MOVL C01618 V=800.0 PL=0
MOVL C01619 V=800.0 PL=0
MOVL C01620 V=800.0 PL=0
MOVL C01621 V=800.0 PL=0
MOVL C01622 V=800.0 PL=0
MOVL C01623 V=800.0 PL=0
MOVL C01624 V=800.0 PL=0
MOVL C01625 V=800.0 PL=0
MOVL C01626 V=800.0 PL=0
MOVL C01627 V=800.0 PL=0
MOVL C01628 V=800.0 PL=0
MOVL C01629 V=800.0 PL=0
MOVL C01630 V=800.0 PL=0
MOVL C01631 V=800.0 PL=0
MOVL C01632 V=800.0 PL=0
MOVL C01633 V=800.0 PL=0
MOVL C01634 V=800.0 PL=0
MOVL C01635 V=800.0 PL=0
MOVL C01636 V=800.0 PL=0
MOVL C01637 V=800.0 PL=0
MOVL C01638 V=800.0 PL=0
MOVL C01639 V=800.0 PL=0
MOVL C01640 V=800.0 PL=0
MOVL C01641 V=800.0 PL=0
MOVL C01642 V=800.0 PL=0
MOVL C01643 V=800.0 PL=0
MOVL C01644 V=800.0 PL=0
MOVL C01645 V=800.0 PL=0
MOVL C01646 V=800.0 PL=0
MOVL C01647 V=800.0 PL=0
MOVL C01648 V=800.0 PL=0
MOVL C01649 V=800.0 PL=0
MOVL C01650 V=800.0 PL=0
MOVL C01651 V=800.0 PL=0
MOVL C01652 V=800.0 PL=0
MOVL C01653 V=800.0 PL=0
MOVL C01654 V=800.0 PL=0
MOVL C01655 V=800.0 PL=0
MOVL C01656 V=800.0 PL=0
MOVL C01657 V=800.0 PL=0
MOVL C01658 V=800.0 PL=0
MOVL C01659 V=800.0 PL=0
MOVL C01660 V=800.0 PL=0
MOVL C01661 V=800.0 PL=0
MOVL C01662 V=800.0 PL=0
MOVL C01663 V=800.0 PL=0
MOVL C01664 V=800.0 PL=0
MOVL C01665 V=800.0 PL=0
MOVL C01666 V=800.0 PL=0
MOVL C01667 V=800.0 PL=0
MOVL C01668 V=800.0 PL=0
MOVL C01669 V=800.0 PL=0
MOVL C01670 V=800.0 PL=0
MOVL C01671 V=800.0 PL=0
MOVL C01672 V=800.0 PL=0
MOVL C01673 V=800.0 PL=0
MOVL C01674 V=800.0 PL=0
MOVL C01675 V=800.0 PL=0
MOVL C01676 V=800.0 PL=0
MOVL C01677 V=800.0 PL=0
MOVL C01678 V=800.0 PL=0
MOVL C01679 V=800.0 PL=0
MOVL C01680 V=800.0 PL=0
MOVL C01681 V=800.0 PL=0
MOVL C01682 V=800.0 PL=0
MOVL C01683 V=800.0 PL=0
MOVL C01684 V=800.0 PL=0
MOVL C01685 V=800.0 PL=0
MOVL C01686 V=800.0 PL=0
MOVL C01687 V=800.0 PL=0
MOVL C01688 V=800.0 PL=0
MOVL C01689 V=800.0 PL=0
MOVL C01690 V=800.0 PL=0
MOVL C01691 V=800.0 PL=0
MOVL C01692 V=800.0 PL=0
MOVL C01693 V=800.0 PL=0
MOVL C01694 V=800.0 PL=0
MOVL C01695 V=800.0 PL=0
MOVL C01696 V=800.0 PL=0
MOVL C01697 V=800.0 PL=0
MOVL C01698 V=800.0 PL=0
MOVL C01699 V=800.0 PL=0
MOVL C01700 V=800.0 PL=0
MOVL C01701 V=800.0 PL=0
MOVL C01702 V=800.0 PL=0
MOVL C01703 V=800.0 PL=0
MOVL C01704 V=800.0 PL=0
MOVL C01705 V=800.0 PL=0
MOVL C01706 V=800.0 PL=0
MOVL C01707 V=800.0 PL=0
MOVL C01708 V=800.0 PL=0
MOVL C01709 V=800.0 PL=0
MOVL C01710 V=800.0 PL=0
MOVL C01711 V=800.0 PL=0
MOVL C01712 V=800.0 PL=0
MOVL C01713 V=800.0 PL=0
MOVL C01714 V=800.0 PL=0
MOVL C01715 V=800.0 PL=0
MOVL C01716 V=800.0 PL=0
MOVL C01717 V=800.0 PL=0
MOVL C01718 V=800.0 PL=0
MOVL C01719 V=800.0 PL=0
MOVL C01720 V=800.0 PL=0
MOVL C01721 V=800.0 PL=0
MOVL C01722 V=800.0 PL=0
MOVL C01723 V=800.0 PL=0
MOVL C01724 V=800.0 PL=0
MOVL C01725 V=800.0 PL=0
MOVL C01726 V=800.0 PL=0
MOVL C01727 V=800.0 PL=0
MOVL C01728 V=800.0 PL=0
MOVL C01729 V=800.0 PL=0
MOVL C01730 V=800.0 PL=0
MOVL C01731 V=800.0 PL=0
MOVL C01732 V=800.0 PL=0
MOVL C01733 V=800.0 PL=0
MOVL C01734 V=800.0 PL=0
MOVL C01735 V=800.0 PL=0
MOVL C01736 V=800.0 PL=0
MOVL C01737 V=800.0 PL=0
MOVL C01738 V=800.0 PL=0
MOVL C01739 V=800.0 PL=0
MOVL C01740 V=800.0 PL=0
MOVL C01741 V=800.0 PL=0
MOVL C01742 V=800.0 PL=0
MOVL C01743 V=800.0 PL=0
MOVL C01744 V=800.0 PL=0
MOVL C01745 V=800.0 PL=0
MOVL C01746 V=800.0 PL=0
MOVL C01747 V=800.0 PL=0
MOVL C01748 V=800.0 PL=0
MOVL C01749 V=800.0 PL=0
MOVL C01750 V=800.0 PL=0
MOVL C01751 V=800.0 PL=0
MOVL C01752 V=800.0 PL=0
MOVL C01753 V=800.0 PL=0
MOVL C01754 V=800.0 PL=0
MOVL C01755 V=800.0 PL=0
MOVL C01756 V=800.0 PL=0
MOVL C01757 V=800.0 PL=0
MOVL C01758 V=800.0 PL=0
MOVL C01759 V=800.0 PL=0
MOVL C01760 V=800.0 PL=0
MOVL C01761 V=800.0 PL=0
MOVL C01762 V=800.0 PL=0
MOVL C01763 V=800.0 PL=0
MOVL C01764 V=800.0 PL=0
MOVL C01765 V=800.0 PL=0
MOVL C01766 V=800.0 PL=0
MOVL C01767 V=800.0 PL=0
MOVL C01768 V=800.0 PL=0
MOVL C01769 V=800.0 PL=0
MOVL C01770 V=800.0 PL=0
MOVL C01771 V=800.0 PL=0
MOVL C01772 V=800.0 PL=0
MOVL C01773 V=800.0 PL=0
MOVL C01774 V=800.0 PL=0
MOVL C01775 V=800.0 PL=0
MOVL C01776 V=800.0 PL=0
MOVL C01777 V=800.0 PL=0
MOVL C01778 V=800.0 PL=0
MOVL C01779 V=800.0 PL=0
MOVL C01780 V=800.0 PL=0
MOVL C01781 V=800.0 PL=0
MOVL C01782 V=800.0 PL=0
MOVL C01783 V=800.0 PL=0
MOVL C01784 V=800.0 PL=0
MOVL C01785 V=800.0 PL=0
MOVL C01786 V=800.0 PL=0
MOVL C01787 V=800.0 PL=0
MOVL C01788 V=800.0 PL=0
MOVL C01789 V=800.0 PL=0
MOVL C01790 V=800.0 PL=0
MOVL C01791 V=800.0 PL=0
MOVL C01792 V=800.0 PL=0
MOVL C01793 V=800.0 PL=0
MOVL C01794 V=800.0 PL=0
MOVL C01795 V=800.0 PL=0
MOVL C01796 V=800.0 PL=0
MOVL C01797 V=800.0 PL=0
MOVL C01798 V=800.0 PL=0
MOVL C01799 V=800.0 PL=0
MOVL C01800 V=800.0 PL=0
MOVL C01801 V=800.0 PL=0
MOVL C01802 V=800.0 PL=0
MOVL C01803 V=800.0 PL=0
MOVL C01804 V=800.0 PL=0
MOVL C01805 V=800.0 PL=0
MOVL C01806 V=800.0 PL=0
MOVL C01807 V=800.0 PL=0
MOVL C01808 V=800.0 PL=0
MOVL C01809 V=800.0 PL=0
MOVL C01810 V=800.0 PL=0
MOVL C01811 V=800.0 PL=0
MOVL C01812 V=800.0 PL=0
MOVL C01813 V=800.0 PL=0
MOVL C01814 V=800.0 PL=0
MOVL C01815 V=800.0 PL=0
MOVL C01816 V=800.0 PL=0
MOVL C01817 V=800.0 PL=0
MOVL C01818 V=800.0 PL=0
MOVL C01819 V=800.0 PL=0
MOVL C01820 V=800.0 PL=0
MOVL C01821 V=800.0 PL=0
MOVL C01822 V=800.0 PL=0
MOVL C01823 V=800.0 PL=0
MOVL C01824 V=800.0 PL=0
MOVL C01825 V=800.0 PL=0
MOVL C01826 V=800.0 PL=0
MOVL C01827 V=800.0 PL=0
MOVL C01828 V=800.0 PL=0
MOVL C01829 V=800.0 PL=0
MOVL C01830 V=800.0 PL=0
MOVL C01831 V=800.0 PL=0
MOVL C01832 V=800.0 PL=0
MOVL C01833 V=800.0 PL=0
MOVL C01834 V=800.0 PL=0
MOVL C01835 V=800.0 PL=0
MOVL C01836 V=800.0 PL=0
MOVL C01837 V=800.0 PL=0
MOVL C01838 V=800.0 PL=0
MOVL C01839 V=800.0 PL=0
MOVL C01840 V=800.0 PL=0
MOVL C01841 V=800.0 PL=0
MOVL C01842 V=800.0 PL=0
MOVL C01843 V=800.0 PL=0
MOVL C01844 V=800.0 PL=0
MOVL C01845 V=800.0 PL=0
MOVL C01846 V=800.0 PL=0
MOVL C01847 V=800.0 PL=0
MOVL C01848 V=800.0 PL=0
MOVL C01849 V=800.0 PL=0
MOVL C01850 V=800.0 PL=0
MOVL C01851 V=800.0 PL=0
MOVL C01852 V=800.0 PL=0
MOVL C01853 V=800.0 PL=0
MOVL C01854 V=800.0 PL=0
MOVL C01855 V=800.0 PL=0
MOVL C01856 V=800.0 PL=0
MOVL C01857 V=800.0 PL=0
MOVL C01858 V=800.0 PL=0
MOVL C01859 V=800.0 PL=0
MOVL C01860 V=800.0 PL=0
MOVL C01861 V=800.0 PL=0
MOVL C01862 V=800.0 PL=0
MOVL C01863 V=800.0 PL=0
MOVL C01864 V=800.0 PL=0
MOVL C01865 V=800.0 PL=0
MOVL C01866 V=800.0 PL=0
MOVL C01867 V=800.0 PL=0
MOVL C01868 V=800.0 PL=0
MOVL C01869 V=800.0 PL=0
MOVL C01870 V=800.0 PL=0
MOVL C01871 V=800.0 PL=0
MOVL C01872 V=800.0 PL=0
MOVL C01873 V=800.0 PL=0
MOVL C01874 V=800.0 PL=0
MOVL C01875 V=800.0 PL=0
MOVL C01876 V=800.0 PL=0
MOVL C01877 V=800.0 PL=0
MOVL C01878 V=800.0 PL=0
MOVL C01879 V=800.0 PL=0
MOVL C01880 V=800.0 PL=0
MOVL C01881 V=800.0 PL=0
MOVL C01882 V=800.0 PL=0
MOVL C01883 V=800.0 PL=0
MOVL C01884 V=800.0 PL=0
MOVL C01885 V=800.0 PL=0
MOVL C01886 V=800.0 PL=0
MOVL C01887 V=800.0 PL=0
MOVL C01888 V=800.0 PL=0
MOVL C01889 V=800.0 PL=0
MOVL C01890 V=800.0 PL=0
MOVL C01891 V=800.0 PL=0
MOVL C01892 V=800.0 PL=0
MOVL C01893 V=800.0 PL=0
MOVL C01894 V=800.0 PL=0
MOVL C01895 V=800.0 PL=0
MOVL C01896 V=800.0 PL=0
MOVL C01897 V=800.0 PL=0
MOVL C01898 V=800.0 PL=0
MOVL C01899 V=800.0 PL=0
MOVL C01900 V=800.0 PL=0
MOVL C01901 V=800.0 PL=0
MOVL C01902 V=800.0 PL=0
MOVL C01903 V=800.0 PL=0
MOVL C01904 V=800.0 PL=0
MOVL C01905 V=800.0 PL=0
MOVL C01906 V=800.0 PL=0
MOVL C01907 V=800.0 PL=0
MOVL C01908 V=800.0 PL=0
MOVL C01909 V=800.0 PL=0
MOVL C01910 V=800.0 PL=0
MOVL C01911 V=800.0 PL=0
MOVL C01912 V=800.0 PL=0
MOVL C01913 V=800.0 PL=0
MOVL C01914 V=800.0 PL=0
MOVL C01915 V=800.0 PL=0
MOVL C01916 V=800.0 PL=0
MOVL C01917 V=800.0 PL=0
MOVL C01918 V=800.0 PL=0
MOVL C01919 V=800.0 PL=0
MOVL C01920 V=800.0 PL=0
MOVL C01921 V=800.0 PL=0
MOVL C01922 V=800.0 PL=0
MOVL C01923 V=800.0 PL=0
MOVL C01924 V=800.0 PL=0
MOVL C01925 V=800.0 PL=0
MOVL C01926 V=800.0 PL=0
MOVL C01927 V=800.0 PL=0
MOVL C01928 V=800.0 PL=0
MOVL C01929 V=800.0 PL=0
MOVL C01930 V=800.0 PL=0
MOVL C01931 V=800.0 PL=0
MOVL C01932 V=800.0 PL=0
MOVL C01933 V=800.0 PL=0
MOVL C01934 V=800.0 PL=0
MOVL C01935 V=800.0 PL=0
MOVL C01936 V=800.0 PL=0
MOVL C01937 V=800.0 PL=0
MOVL C01938 V=800.0 PL=0
MOVL C01939 V=800.0 PL=0
MOVL C01940 V=800.0 PL=0
MOVL C01941 V=800.0 PL=0
MOVL C01942 V=800.0 PL=0
MOVL C01943 V=800.0 PL=0
MOVL C01944 V=800.0 PL=0
MOVL C01945 V=800.0 PL=0
MOVL C01946 V=800.0 PL=0
MOVL C01947 V=800.0 PL=0
MOVL C01948 V=800.0 PL=0
MOVL C01949 V=800.0 PL=0
MOVL C01950 V=800.0 PL=0
MOVL C01951 V=800.0 PL=0
MOVL C01952 V=800.0 PL=0
MOVL C01953 V=800.0 PL=0
MOVL C01954 V=800.0 PL=0
MOVL C01955 V=800.0 PL=0
MOVL C01956 V=800.0 PL=0
MOVL C01957 V=800.0 PL=0
MOVL C01958 V=800.0 PL=0
MOVL C01959 V=800.0 PL=0
MOVL C01960 V=800.0 PL=0
MOVL C01961 V=800.0 PL=0
MOVL C01962 V=800.0 PL=0
MOVL C01963 V=800.0 PL=0
MOVL C01964 V=800.0 PL=0
MOVL C01965 V=800.0 PL=0
MOVL C01966 V=800.0 PL=0
MOVL C01967 V=800.0 PL=0
MOVL C01968 V=800.0 PL=0
MOVL C01969 V=800.0 PL=0
MOVL C01970 V=800.0 PL=0
MOVL C01971 V=800.0 PL=0
MOVL C01972 V=800.0 PL=0
MOVL C01973 V=800.0 PL=0
MOVL C01974 V=800.0 PL=0
MOVL C01975 V=800.0 PL=0
MOVL C01976 V=800.0 PL=0
MOVL C01977 V=800.0 PL=0
MOVL C01978 V=800.0 PL=0
MOVL C01979 V=800.0 PL=0
MOVL C01980 V=800.0 PL=0
MOVL C01981 V=800.0 PL=0
MOVL C01982 V=800.0 PL=0
MOVL C01983 V=800.0 PL=0
MOVL C01984 V=800.0 PL=0
MOVL C01985 V=800.0 PL=0
MOVL C01986 V=800.0 PL=0
MOVL C01987 V=800.0 PL=0
MOVL C01988 V=800.0 PL=0
MOVL C01989 V=800.0 PL=0
MOVL C01990 V=800.0 PL=0
MOVL C01991 V=800.0 PL=0
MOVL C01992 V=800.0 PL=0
MOVL C01993 V=800.0 PL=0
MOVL C01994 V=800.0 PL=0
MOVL C01995 V=800.0 PL=0
MOVL C01996 V=800.0 PL=0
MOVL C01997 V=800.0 PL=0
MOVL C01998 V=800.0 PL=0
MOVL C01999 V=800.0 PL=0
MOVL C02000 V=800.0 PL=0
MOVL C02001 V=800.0 PL=0
MOVL C02002 V=800.0 PL=0
MOVL C02003 V=800.0 PL=0
MOVL C02004 V=800.0 PL=0
MOVL C02005 V=800.0 PL=0
MOVL C02006 V=800.0 PL=0
MOVL C02007 V=800.0 PL=0
MOVL C02008 V=800.0 PL=0
MOVL C02009 V=800.0 PL=0
MOVL C02010 V=800.0 PL=0
MOVL C02011 V=800.0 PL=0
MOVL C02012 V=800.0 PL=0
MOVL C02013 V=800.0 PL=0
MOVL C02014 V=800.0 PL=0
MOVL C02015 V=800.0 PL=0
MOVL C02016 V=800.0 PL=0
MOVL C02017 V=800.0 PL=0
MOVL C02018 V=800.0 PL=0
MOVL C02019 V=800.0 PL=0
MOVL C02020 V=800.0 PL=0
MOVL C02021 V=800.0 PL=0
MOVL C02022 V=800.0 PL=0
MOVL C02023 V=800.0 PL=0
MOVL C02024 V=800.0 PL=0
MOVL C02025 V=800.0 PL=0
MOVL C02026 V=800.0 PL=0
MOVL C02027 V=800.0 PL=0
MOVL C02028 V=800.0 PL=0
MOVL C02029 V=800.0 PL=0
MOVL C02030 V=800.0 PL=0
MOVL C02031 V=800.0 PL=0
MOVL C02032 V=800.0 PL=0
MOVL C02033 V=800.0 PL=0
MOVL C02034 V=800.0 PL=0
MOVL C02035 V=800.0 PL=0
MOVL C02036 V=800.0 PL=0
MOVL C02037 V=800.0 PL=0
MOVL C02038 V=800.0 PL=0
MOVL C02039 V=800.0 PL=0
